// Functions/Image Filtering/F_VN_FillHoles

	{attribute 'TcIecLibraryType'}
	{attribute 'external_name' := 'F_VN_FillHoles_GUID_45C31AD9_EBC0_4725_EDA8_84DF2214AC65'}
	(* Fill holes within a gray-scale single-channel image. (equivalent to finding dark border objects) *)
	FUNCTION F_VN_FillHoles : HRESULT
	VAR_INPUT
		ipSrcImage	:	ITcVnImage;	(* Source image (USINT, UINT, INT, REAL, or LREAL, 1 channel) *)
		ipDestImage	:	REFERENCE TO ITcVnImage;	(* Destination image (An appropriate destination image will be created if required.) *)
		hrPrev	:	HRESULT;	(* HRESULT indicating the result of previous operations (If SUCCEEDED(hrPrev) equals false, no operation is executed.) *)
	END_VAR

END_FUNCTION

// Functions/Image Filtering/F_VN_GaussianFilter

	{attribute 'TcIecLibraryType'}
	{attribute 'external_name' := 'F_VN_GaussianFilter_GUID_95A7A389_C35E_4A28_C080_30D43CAAA1FC'}
	(* Apply a Gaussian filter to smooth the image. *)
	FUNCTION F_VN_GaussianFilter : HRESULT
	VAR_INPUT
		ipSrcImage	:	ITcVnImage;	(* Source image *)
		ipDestImage	:	REFERENCE TO ITcVnImage;	(* Destination image (An appropriate destination image will be created if required.) *)
		nFilterWidth	:	UDINT;	(* Filter width in pixels (1, 3, 5, 7, ...) *)
		nFilterHeight	:	UDINT;	(* Filter height in pixels (1, 3, 5, 7, ...) *)
		hrPrev	:	HRESULT;	(* HRESULT indicating the result of previous operations (If SUCCEEDED(hrPrev) equals false, no operation is executed.) *)
	END_VAR

END_FUNCTION

// Functions/Image Filtering/F_VN_GaussianFilterExp

	{attribute 'TcIecLibraryType'}
	{attribute 'external_name' := 'F_VN_GaussianFilterExp_GUID_44AEB57C_BFD9_4E61_C3CD_471B6E3D0B02'}
	(* Apply a Gaussian filter to smooth the image. (expert function) *)
	FUNCTION F_VN_GaussianFilterExp : HRESULT
	VAR_INPUT
		ipSrcImage	:	ITcVnImage;	(* Source image *)
		ipDestImage	:	REFERENCE TO ITcVnImage;	(* Destination image (An appropriate destination image will be created if required.) *)
		nFilterWidth	:	UDINT;	(* Filter width in pixels (1, 3, 5, 7, ...) *)
		nFilterHeight	:	UDINT;	(* Filter height in pixels (1, 3, 5, 7, ...) *)
		fSigmaX	:	LREAL;	(* Gaussian kernel standard deviation in X direction (>= 0, automatically chosen if 0) *)
		fSigmaY	:	LREAL;	(* Gaussian kernel standard deviation in Y direction (>= 0, automatically chosen if 0) *)
		eBorderType	:	ETcVnBorderInterpolationMethod;	(* Image border handling *)
		hrPrev	:	HRESULT;	(* HRESULT indicating the result of previous operations (If SUCCEEDED(hrPrev) equals false, no operation is executed.) *)
	END_VAR

END_FUNCTION

// Functions/Image Filtering/F_VN_LaplacianFilter

	{attribute 'TcIecLibraryType'}
	{attribute 'external_name' := 'F_VN_LaplacianFilter_GUID_22F6738F_8883_4E9E_FB58_F8CB0A9D323F'}
	(* Apply a Laplacian filter to an image. *)
	FUNCTION F_VN_LaplacianFilter : HRESULT
	VAR_INPUT
		ipSrcImage	:	ITcVnImage;	(* Source image *)
		ipDestImage	:	REFERENCE TO ITcVnImage;	(* Destination image (An appropriate destination image will be created if required.) *)
		eDestDepth	:	ETcVnElementType;	(* Destination image depth *)
		hrPrev	:	HRESULT;	(* HRESULT indicating the result of previous operations (If SUCCEEDED(hrPrev) equals false, no operation is executed.) *)
	END_VAR

END_FUNCTION

// Functions/Image Filtering/F_VN_LaplacianFilterExp

	{attribute 'TcIecLibraryType'}
	{attribute 'external_name' := 'F_VN_LaplacianFilterExp_GUID_80C0BC32_CA68_4BC2_FC4E_748676C48192'}
	(* Apply a Laplacian filter to an image. (expert function) *)
	FUNCTION F_VN_LaplacianFilterExp : HRESULT
	VAR_INPUT
		ipSrcImage	:	ITcVnImage;	(* Source image *)
		ipDestImage	:	REFERENCE TO ITcVnImage;	(* Destination image (An appropriate destination image will be created if required.) *)
		eDestDepth	:	ETcVnElementType;	(* Destination image depth *)
		nKernelSize	:	UDINT;	(* Aperture size used to compute the second-derivative filters (1, 3, 5, ..., 31) *)
		fScale	:	LREAL;	(* Scale factor for the computed derivative values *)
		fDelta	:	LREAL;	(* Delta value that is added to the results before storing them *)
		eBorderType	:	ETcVnBorderInterpolationMethod;	(* Image border handling *)
		hrPrev	:	HRESULT;	(* HRESULT indicating the result of previous operations (If SUCCEEDED(hrPrev) equals false, no operation is executed.) *)
	END_VAR

END_FUNCTION

// Functions/Image Filtering/F_VN_LocalMaxima

	{attribute 'TcIecLibraryType'}
	{attribute 'external_name' := 'F_VN_LocalMaxima_GUID_037C572B_82DC_43A0_C6A2_016E37C2D982'}
	(* Find local maxima in a gray-scale single-channel image. The found maxima are marked by a value of 1 in the destination image. *)
	FUNCTION F_VN_LocalMaxima : HRESULT
	VAR_INPUT
		ipSrcImage	:	ITcVnImage;	(* Source image (USINT or UINT, 1 channel) *)
		ipDestImage	:	REFERENCE TO ITcVnImage;	(* Destination image (Must be different from ipSrcImage! An appropriate destination image will be created if required.) *)
		hrPrev	:	HRESULT;	(* HRESULT indicating the result of previous operations (If SUCCEEDED(hrPrev) equals false, no operation is executed.) *)
	END_VAR

END_FUNCTION

// Functions/Image Filtering/F_VN_LocalMinima

	{attribute 'TcIecLibraryType'}
	{attribute 'external_name' := 'F_VN_LocalMinima_GUID_332C39B6_195E_4830_D66F_8C7BE687196D'}
	(* Find local minima in a gray-scale single-channel image. The found minima are marked by a value of 1 in the destination image. *)
	FUNCTION F_VN_LocalMinima : HRESULT
	VAR_INPUT
		ipSrcImage	:	ITcVnImage;	(* Source image (USINT or UINT, 1 channel) *)
		ipDestImage	:	REFERENCE TO ITcVnImage;	(* Destination image (Must be different from ipSrcImage! An appropriate destination image will be created if required.) *)
		hrPrev	:	HRESULT;	(* HRESULT indicating the result of previous operations (If SUCCEEDED(hrPrev) equals false, no operation is executed.) *)
	END_VAR

END_FUNCTION

// Functions/Image Filtering/F_VN_MedianFilter

	{attribute 'TcIecLibraryType'}
	{attribute 'external_name' := 'F_VN_MedianFilter_GUID_183F28CD_813D_43D0_CDC8_13AA290F7025'}
	(* Apply a Median filter to an image. *)
	FUNCTION F_VN_MedianFilter : HRESULT
	VAR_INPUT
		ipSrcImage	:	ITcVnImage;	(* Source image (for nFilterSize 3 or 5: USINT, UINT, REAL. For bigger filters, only USINT is supported. *)
		ipDestImage	:	REFERENCE TO ITcVnImage;	(* Destination image (An appropriate destination image will be created if required.) *)
		nFilterSize	:	UDINT;	(* Size (width and height) of the filter (3, 5, 7, ...) *)
		hrPrev	:	HRESULT;	(* HRESULT indicating the result of previous operations (If SUCCEEDED(hrPrev) equals false, no operation is executed.) *)
	END_VAR

END_FUNCTION

// Functions/Image Filtering/F_VN_MorphologicalOperator

	{attribute 'TcIecLibraryType'}
	{attribute 'external_name' := 'F_VN_MorphologicalOperator_GUID_B23434BD_E36C_4E02_E145_B2ED6C6CC2A2'}
	(* Apply a morphological operator. *)
	FUNCTION F_VN_MorphologicalOperator : HRESULT
	VAR_INPUT
		ipSrcImage	:	ITcVnImage;	(* Source image (only 1 channel supported for reconstruction operators) *)
		ipDestImage	:	REFERENCE TO ITcVnImage;	(* Destination image (An appropriate destination image will be created if required.) *)
		eOperator	:	ETcVnMorphologicalOperator;	(* Operator type *)
		ipStructuringElement	:	ITcVnImage;	(* Structuring element to be applied (Typically created via F_VN_CreateStructuringElement.) *)
		hrPrev	:	HRESULT;	(* HRESULT indicating the result of previous operations (If SUCCEEDED(hrPrev) equals false, no operation is executed.) *)
	END_VAR

END_FUNCTION

// Functions/Image Filtering/F_VN_RemoveLocalMaxima

	{attribute 'TcIecLibraryType'}
	{attribute 'external_name' := 'F_VN_RemoveLocalMaxima_GUID_63A5ADDB_B6C9_4B05_E1FA_40A640049502'}
	(* Remove local maxima up to a given height from a gray-scale single-channel image. *)
	FUNCTION F_VN_RemoveLocalMaxima : HRESULT
	VAR_INPUT
		ipSrcImage	:	ITcVnImage;	(* Source image (USINT, UINT, INT, REAL, or LREAL, 1 channel) *)
		ipDestImage	:	REFERENCE TO ITcVnImage;	(* Destination image (An appropriate destination image will be created if required.) *)
		fHeight	:	LREAL;	(* Maximum height of the maxima to be removed (must be greater than 0) *)
		hrPrev	:	HRESULT;	(* HRESULT indicating the result of previous operations (If SUCCEEDED(hrPrev) equals false, no operation is executed.) *)
	END_VAR

END_FUNCTION

// Functions/Image Filtering/F_VN_RemoveLocalMinima

	{attribute 'TcIecLibraryType'}
	{attribute 'external_name' := 'F_VN_RemoveLocalMinima_GUID_D50AAA78_D3B9_408D_D404_A332605EC262'}
	(* Remove local minima up to a given height from a gray-scale single-channel image. *)
	FUNCTION F_VN_RemoveLocalMinima : HRESULT
	VAR_INPUT
		ipSrcImage	:	ITcVnImage;	(* Source image (USINT, UINT, INT, REAL, or LREAL, 1 channel) *)
		ipDestImage	:	REFERENCE TO ITcVnImage;	(* Destination image (An appropriate destination image will be created if required.) *)
		fHeight	:	LREAL;	(* Maximum height of the minima to be removed (must be greater than 0) *)
		hrPrev	:	HRESULT;	(* HRESULT indicating the result of previous operations (If SUCCEEDED(hrPrev) equals false, no operation is executed.) *)
	END_VAR

END_FUNCTION

// Functions/Image Filtering/F_VN_ScharrFilter

	{attribute 'TcIecLibraryType'}
	{attribute 'external_name' := 'F_VN_ScharrFilter_GUID_4C4A4FDA_AE3C_464A_CF07_94424B3EAEFE'}
	(* Calculates the first order derivative in x or y direction using a Scharr filter. *)
	FUNCTION F_VN_ScharrFilter : HRESULT
	VAR_INPUT
		ipSrcImage	:	ITcVnImage;	(* Source image *)
		ipDestImage	:	REFERENCE TO ITcVnImage;	(* Destination image (An appropriate destination image will be created if required.) *)
		eDestDepth	:	ETcVnElementType;	(* Destination image depth *)
		eFilterDirection	:	ETcVnFilterDirection;	(* Filter direction *)
		hrPrev	:	HRESULT;	(* HRESULT indicating the result of previous operations (If SUCCEEDED(hrPrev) equals false, no operation is executed.) *)
	END_VAR

END_FUNCTION

// Functions/Image Filtering/F_VN_ScharrFilterExp

	{attribute 'TcIecLibraryType'}
	{attribute 'external_name' := 'F_VN_ScharrFilterExp_GUID_6408ADDC_C84A_4DA3_CB0C_8C03DB762CD6'}
	(* Calculates the first order derivative in x or y direction using a Scharr filter. (expert function) *)
	FUNCTION F_VN_ScharrFilterExp : HRESULT
	VAR_INPUT
		ipSrcImage	:	ITcVnImage;	(* Source image *)
		ipDestImage	:	REFERENCE TO ITcVnImage;	(* Destination image (An appropriate destination image will be created if required.) *)
		eDestDepth	:	ETcVnElementType;	(* Destination image depth *)
		eFilterDirection	:	ETcVnFilterDirection;	(* Filter direction *)
		fScale	:	LREAL;	(* Scale factor for the computed derivative values *)
		fDelta	:	LREAL;	(* Delta value that is added to the results prior to storing them in dest *)
		eBorderType	:	ETcVnBorderInterpolationMethod;	(* Image border handling *)
		hrPrev	:	HRESULT;	(* HRESULT indicating the result of previous operations (If SUCCEEDED(hrPrev) equals false, no operation is executed.) *)
	END_VAR

END_FUNCTION

// Functions/Image Filtering/F_VN_SeparableCustomFilter

	{attribute 'TcIecLibraryType'}
	{attribute 'external_name' := 'F_VN_SeparableCustomFilter_GUID_1310DFB7_D59D_44ED_EDCE_83E1B6FDCC84'}
	(* Apply a separable custom filter to the image. *)
	FUNCTION F_VN_SeparableCustomFilter : HRESULT
	VAR_INPUT
		ipSrcImage	:	ITcVnImage;	(* Source image *)
		ipDestImage	:	REFERENCE TO ITcVnImage;	(* Destination image (An appropriate destination image will be created if required.) *)
		eDestDepth	:	ETcVnElementType;	(* Destination image depth *)
	END_VAR
	VAR_IN_OUT
		stKernelX	:	TcVnMatrix;	(* 1D custom row-filter kernel with values of type REAL or LREAL *)
		stKernelY	:	TcVnMatrix;	(* 1D custom column-filter kernel with values of type REAL or LREAL *)
	END_VAR
	VAR_INPUT
		hrPrev	:	HRESULT;	(* HRESULT indicating the result of previous operations (If SUCCEEDED(hrPrev) equals false, no operation is executed.) *)
	END_VAR

END_FUNCTION

// Functions/Image Filtering/F_VN_SeparableCustomFilterExp

	{attribute 'TcIecLibraryType'}
	{attribute 'external_name' := 'F_VN_SeparableCustomFilterExp_GUID_BCC4F12D_D44C_4679_C6D6_F7CE17C8407A'}
	(* Apply a separable custom filter to the image. (expert function) *)
	FUNCTION F_VN_SeparableCustomFilterExp : HRESULT
	VAR_INPUT
		ipSrcImage	:	ITcVnImage;	(* Source image *)
		ipDestImage	:	REFERENCE TO ITcVnImage;	(* Destination image (An appropriate destination image will be created if required.) *)
		eDestDepth	:	ETcVnElementType;	(* Destination image depth *)
	END_VAR
	VAR_IN_OUT
		stKernelX	:	TcVnMatrix;	(* 1D custom row-filter kernel with values of type REAL or LREAL *)
		stKernelY	:	TcVnMatrix;	(* 1D custom column-filter kernel with values of type REAL or LREAL *)
		aAnchor	:	TcVnPoint;	(* Anchor point of the kernel *)
	END_VAR
	VAR_INPUT
		fDelta	:	LREAL;	(* Value added to each pixel after filtering *)
		eBorderType	:	ETcVnBorderInterpolationMethod;	(* Image border handling *)
		hrPrev	:	HRESULT;	(* HRESULT indicating the result of previous operations (If SUCCEEDED(hrPrev) equals false, no operation is executed.) *)
	END_VAR

END_FUNCTION

// Functions/Image Filtering/F_VN_SobelFilter

	{attribute 'TcIecLibraryType'}
	{attribute 'external_name' := 'F_VN_SobelFilter_GUID_082961EA_2A54_4C56_CFFB_604B528A29B1'}
	(* Calculates the first, second, or mixed image derivatives using an extended Sobel filter. *)
	FUNCTION F_VN_SobelFilter : HRESULT
	VAR_INPUT
		ipSrcImage	:	ITcVnImage;	(* Source image *)
		ipDestImage	:	REFERENCE TO ITcVnImage;	(* Destination image (An appropriate destination image will be created if required.) *)
		eDestDepth	:	ETcVnElementType;	(* Destination image depth *)
		nXOrder	:	UDINT;	(* Order of the x-derivative (0, 1, 2) *)
		nYOrder	:	UDINT;	(* Order of the y-derivative (0, 1, 2) *)
		hrPrev	:	HRESULT;	(* HRESULT indicating the result of previous operations (If SUCCEEDED(hrPrev) equals false, no operation is executed.) *)
	END_VAR

END_FUNCTION

// Functions/Image Filtering/F_VN_SobelFilterExp

	{attribute 'TcIecLibraryType'}
	{attribute 'external_name' := 'F_VN_SobelFilterExp_GUID_8B414AB6_412D_41C9_E4E5_57ECB320A706'}
	(* Calculates the first, second, third, or mixed image derivatives using an extended Sobel filter. (expert function) *)
	FUNCTION F_VN_SobelFilterExp : HRESULT
	VAR_INPUT
		ipSrcImage	:	ITcVnImage;	(* Source image *)
		ipDestImage	:	REFERENCE TO ITcVnImage;	(* Destination image (An appropriate destination image will be created if required.) *)
		eDestDepth	:	ETcVnElementType;	(* Destination image depth *)
		nXOrder	:	UDINT;	(* Order of the x-derivative (must be < nKernelSize) *)
		nYOrder	:	UDINT;	(* Order of the y-derivative (must be < nKernelSize) *)
		nKernelSize	:	UDINT;	(* Size of the extended Sobel kernel (3, 5, 7, ..., 31) *)
		fScale	:	LREAL;	(* Scale factor for the computed derivative values *)
		fDelta	:	LREAL;	(* Delta value that is added to the results prior to storing them in dest *)
		eBorderType	:	ETcVnBorderInterpolationMethod;	(* Image border handling *)
		hrPrev	:	HRESULT;	(* HRESULT indicating the result of previous operations (If SUCCEEDED(hrPrev) equals false, no operation is executed.) *)
	END_VAR

END_FUNCTION

// Functions/Image Filtering/F_VN_VarianceFilter

	{attribute 'TcIecLibraryType'}
	{attribute 'external_name' := 'F_VN_VarianceFilter_GUID_02C328AD_BE75_4B70_DC76_31CB3237B1CA'}
	(* Calculates the local variance of an image. *)
	FUNCTION F_VN_VarianceFilter : HRESULT
	VAR_INPUT
		ipSrcImage	:	ITcVnImage;	(* Source image. Only TCVN_ET_USINT Type is supported.  *)
		ipDestImage	:	REFERENCE TO ITcVnImage;	(* Destination image of type TCVN_ET_UINT (An appropriate destination image will be created if required.) *)
		nKernelSize	:	UDINT;	(* Size of the kernel *)
		hrPrev	:	HRESULT;	(* HRESULT indicating the result of previous operations (If SUCCEEDED(hrPrev) equals false, no operation is executed.) *)
	END_VAR

END_FUNCTION

// Functions/Image Filtering/F_VN_VarianceFilterExp

	{attribute 'TcIecLibraryType'}
	{attribute 'external_name' := 'F_VN_VarianceFilterExp_GUID_48CB282B_6C36_4355_F8DD_C52CAA374075'}
	(* Calculates the local variance of an image. (expert function) *)
	FUNCTION F_VN_VarianceFilterExp : HRESULT
	VAR_INPUT
		ipSrcImage	:	ITcVnImage;	(* Source image. Only TCVN_ET_USINT Type is supported. *)
		ipDestImage	:	REFERENCE TO ITcVnImage;	(* Destination image of type TCVN_ET_UINT (An appropriate destination image will be created if required.) *)
		nKernelSize	:	UDINT;	(* Size of the kernel *)
		fScale	:	LREAL;	(* Scale factor for the computed variance values *)
		eBorderType	:	ETcVnBorderInterpolationMethod;	(* Image border handling *)
		hrPrev	:	HRESULT;	(* HRESULT indicating the result of previous operations (If SUCCEEDED(hrPrev) equals false, no operation is executed.) *)
	END_VAR

END_FUNCTION

// Functions/Miscellaneous/F_VN_CheckFunctionInitialization

	{attribute 'TcIecLibraryType'}
	{attribute 'external_name' := 'F_VN_CheckFunctionInitialization_GUID_2C8223A2_77FF_41C2_DA7B_831BEC82D7D0'}
	(* Check if a function is initialized with the specified options. *)
	FUNCTION F_VN_CheckFunctionInitialization : HRESULT
	VAR_INPUT
		eFunction	:	ETcVnInitializableFunction;	(* Initializable function *)
		nOptions	:	ULINT;	(* Initialization options for the function *)
		hrPrev	:	HRESULT;	(* HRESULT indicating the result of previous operations (If SUCCEEDED(hrPrev) equals false, no operation is executed.) *)
	END_VAR

END_FUNCTION

// Functions/Miscellaneous/F_VN_ClipLineToBoundary

	{attribute 'TcIecLibraryType'}
	{attribute 'external_name' := 'F_VN_ClipLineToBoundary_GUID_B482B9AE_8531_4446_C981_B7F9A09BE1A0'}
	(* Clips a line to a rectangular boundary. *)
	FUNCTION F_VN_ClipLineToBoundary : HRESULT
	VAR_IN_OUT
		aLine	:	TcVnVector4_LREAL;	(* The first and second element describe the x and y component of the direction vector. The third and fourth element describe the x and y component of the position vector. *)
	END_VAR
	VAR_INPUT
		nX1	:	DINT;	(* x of top left rectangle point *)
		nY1	:	DINT;	(* y of top left rectangle point *)
		nX2	:	DINT;	(* x of bottom right rectangle point *)
		nY2	:	DINT;	(* Y of bottom right rectangle point *)
	END_VAR
	VAR_IN_OUT
		aStartPoint	:	TcVnPoint2_REAL;	(* Returns the clipped starting point of the line. *)
		aEndPoint	:	TcVnPoint2_REAL;	(* Returns the clipped end point of the line. *)
	END_VAR
	VAR_INPUT
		hrPrev	:	HRESULT;	(* HRESULT indicating the result of previous operations (If SUCCEEDED(hrPrev) equals false, no operation is executed.) *)
	END_VAR

END_FUNCTION

// Functions/Miscellaneous/F_VN_ClipLineToBoundary_ITcVnImage

	{attribute 'TcIecLibraryType'}
	{attribute 'external_name' := 'F_VN_ClipLineToBoundary_ITcVnImage_GUID_0FCA2B5E_8797_43C5_D314_057DDEA9B856'}
	(* Clips a line to the boundary of an image. *)
	FUNCTION F_VN_ClipLineToBoundary_ITcVnImage : HRESULT
	VAR_IN_OUT
		aLine	:	TcVnVector4_LREAL;	(* The first and second element describe the x and y component of the direction vector. The third and fourth element describe the x and y component of the position vector. *)
	END_VAR
	VAR_INPUT
		ipImage	:	ITcVnImage;	(* Image, from which to derive the boundary *)
	END_VAR
	VAR_IN_OUT
		aStartPoint	:	TcVnPoint2_REAL;	(* Returns the clipped starting point of the line. *)
		aEndPoint	:	TcVnPoint2_REAL;	(* Returns the clipped end point of the line. *)
	END_VAR
	VAR_INPUT
		hrPrev	:	HRESULT;	(* HRESULT indicating the result of previous operations (If SUCCEEDED(hrPrev) equals false, no operation is executed.) *)
	END_VAR

END_FUNCTION

// Functions/Miscellaneous/F_VN_ClipLineToBoundary_TcVnRectangle_DINT

	{attribute 'TcIecLibraryType'}
	{attribute 'external_name' := 'F_VN_ClipLineToBoundary_TcVnRectangle_DINT_GUID_6C0A9627_1BE4_42B6_C7E1_34156AEEC835'}
	(* Clips a line to a rectangular boundary. *)
	FUNCTION F_VN_ClipLineToBoundary_TcVnRectangle_DINT : HRESULT
	VAR_IN_OUT
		aLine	:	TcVnVector4_LREAL;	(* The first and second element describe the x and y component of the direction vector. The third and fourth element describe the x and y component of the position vector. *)
		stRectangle	:	TcVnRectangle_DINT;	(* Rectangular boundary *)
		aStartPoint	:	TcVnPoint2_REAL;	(* Returns the clipped starting point of the line. *)
		aEndPoint	:	TcVnPoint2_REAL;	(* Returns the clipped end point of the line. *)
	END_VAR
	VAR_INPUT
		hrPrev	:	HRESULT;	(* HRESULT indicating the result of previous operations (If SUCCEEDED(hrPrev) equals false, no operation is executed.) *)
	END_VAR

END_FUNCTION

// Functions/Miscellaneous/F_VN_ConvertITcUnknownToITcVnBitmapExport

	{attribute 'TcIecLibraryType'}
	{attribute 'external_name' := 'F_VN_ConvertITcUnknownToITcVnBitmapExport_GUID_C5AC5150_1991_4233_D664_F885FA18923A'}
	(* Convert an ITcUnknown interface pointer to an ITcVnBitmapExport interface pointer. The destination pointer will be released (if existing) and set to the source pointer. The source pointer will be set to 0. *)
	FUNCTION F_VN_ConvertITcUnknownToITcVnBitmapExport : HRESULT
	VAR_INPUT
		ipSrc	:	REFERENCE TO ITcUnknown;	(* Source pointer *)
		ipDest	:	REFERENCE TO ITcVnBitmapExport;	(* Destination pointer *)
		hrPrev	:	HRESULT;	(* HRESULT indicating the result of previous operations (If SUCCEEDED(hrPrev) equals false, no operation is executed.) *)
	END_VAR

END_FUNCTION

// Functions/Miscellaneous/F_VN_ConvertITcUnknownToITcVnContainer

	{attribute 'TcIecLibraryType'}
	{attribute 'external_name' := 'F_VN_ConvertITcUnknownToITcVnContainer_GUID_F89008A1_7EE5_44B8_ED7B_BAB16CAC9C5B'}
	(* Convert an ITcUnknown interface pointer to an ITcVnContainer interface pointer. The destination pointer will be released (if existing) and set to the source pointer. The source pointer will be set to 0. *)
	FUNCTION F_VN_ConvertITcUnknownToITcVnContainer : HRESULT
	VAR_INPUT
		ipSrc	:	REFERENCE TO ITcUnknown;	(* Source pointer *)
		ipDest	:	REFERENCE TO ITcVnContainer;	(* Destination pointer *)
		hrPrev	:	HRESULT;	(* HRESULT indicating the result of previous operations (If SUCCEEDED(hrPrev) equals false, no operation is executed.) *)
	END_VAR

END_FUNCTION

// Functions/Miscellaneous/F_VN_ConvertITcUnknownToITcVnImage

	{attribute 'TcIecLibraryType'}
	{attribute 'external_name' := 'F_VN_ConvertITcUnknownToITcVnImage_GUID_F768478E_506F_4CE2_C2D1_8F48D5018F3E'}
	(* Convert an ITcUnknown interface pointer to an ITcVnImage interface pointer. The destination pointer will be released (if existing) and set to the source pointer. The source pointer will be set to 0. *)
	FUNCTION F_VN_ConvertITcUnknownToITcVnImage : HRESULT
	VAR_INPUT
		ipSrc	:	REFERENCE TO ITcUnknown;	(* Source pointer *)
		ipDest	:	REFERENCE TO ITcVnImage;	(* Destination pointer *)
		hrPrev	:	HRESULT;	(* HRESULT indicating the result of previous operations (If SUCCEEDED(hrPrev) equals false, no operation is executed.) *)
	END_VAR

END_FUNCTION

// Functions/Miscellaneous/F_VN_ConvertITcUnknownToITcVnMlModel

	{attribute 'TcIecLibraryType'}
	{attribute 'external_name' := 'F_VN_ConvertITcUnknownToITcVnMlModel_GUID_EBE69EF4_1DE6_4A53_D37C_0D2CB88EB72B'}
	(* Convert an ITcUnknown interface pointer to an ITcVnMlModel interface pointer. The destination pointer will be released (if existing) and set to the source pointer. The source pointer will be set to 0. *)
	FUNCTION F_VN_ConvertITcUnknownToITcVnMlModel : HRESULT
	VAR_INPUT
		ipSrc	:	REFERENCE TO ITcUnknown;	(* Source pointer *)
		ipDest	:	REFERENCE TO ITcVnMlModel;	(* Destination pointer *)
		hrPrev	:	HRESULT;	(* HRESULT indicating the result of previous operations (If SUCCEEDED(hrPrev) equals false, no operation is executed.) *)
	END_VAR

END_FUNCTION

// Functions/Miscellaneous/F_VN_DeinitializeFunction

	{attribute 'TcIecLibraryType'}
	{attribute 'external_name' := 'F_VN_DeinitializeFunction_GUID_D1F3361E_3ED0_4425_EAC1_FD419D650FCA'}
	(* Deinitialize the specified options for the function. *)
	FUNCTION F_VN_DeinitializeFunction : HRESULT
	VAR_INPUT
		eFunction	:	ETcVnInitializableFunction;	(* Initializable function *)
		nOptions	:	ULINT;	(* Initialization options for the function *)
		hrPrev	:	HRESULT;	(* HRESULT indicating the result of previous operations (If SUCCEEDED(hrPrev) equals false, no operation is executed.) *)
	END_VAR

END_FUNCTION

// Functions/Miscellaneous/F_VN_GetTimestamp

	{attribute 'TcIecLibraryType'}
	{attribute 'external_name' := 'F_VN_GetTimestamp_GUID_2D68E61A_B781_405D_F127_30855B02D50E'}
	(* Get the timestamp (actual DC time) from the last change of an object (e.g. ITcVnImage or ITcVnContainer) *)
	FUNCTION F_VN_GetTimestamp : HRESULT
	VAR_INPUT
		ipUnknown	:	ITcUnknown;	(* An object implementing ITcUnknown and ITcVnTimestamp (e.g. ITcVnImage or ITcVnContainer) *)
	END_VAR
	VAR_IN_OUT
		nTimestamp	:	LINT;	(* Returns the timestamp *)
	END_VAR
	VAR_INPUT
		hrPrev	:	HRESULT;	(* HRESULT indicating the result of previous operations (If SUCCEEDED(hrPrev) equals false, no operation is executed.) *)
	END_VAR

END_FUNCTION

// Functions/Miscellaneous/F_VN_HuMomentInvariants

	{attribute 'TcIecLibraryType'}
	{attribute 'external_name' := 'F_VN_HuMomentInvariants_GUID_578FD112_2DC5_4CAD_F1B3_F670083C2AF6'}
	(* Computes the Hu moment invariants. *)
	FUNCTION F_VN_HuMomentInvariants : HRESULT
	VAR_IN_OUT
		stMoments	:	TcVnMoments;	(* Moments from which to compute the Hu invariants *)
		aHuInvariants	:	TcVnArray7_LREAL;	(* Returns the Hu moment invariants *)
	END_VAR
	VAR_INPUT
		hrPrev	:	HRESULT;	(* HRESULT indicating the result of previous operations (If SUCCEEDED(hrPrev) equals false, no operation is executed.) *)
	END_VAR

END_FUNCTION

// Functions/Miscellaneous/F_VN_InitMatrixStruct

	{attribute 'TcIecLibraryType'}
	{attribute 'external_name' := 'F_VN_InitMatrixStruct_GUID_6C97114E_1940_4DE0_F672_C2C518D51A5C'}
	(* Initialize a struct of the type TcVnMatrix extending a buffer with metainformation so that it can be used as a matrix. *)
	FUNCTION F_VN_InitMatrixStruct : HRESULT
	VAR_INPUT
		pSrcBuffer	:	PVOID;	(* Source buffer *)
	END_VAR
	VAR_IN_OUT
		stDestMatrix	:	TcVnMatrix;	(* Returns completed matrix struct *)
	END_VAR
	VAR_INPUT
		nRows	:	UDINT;	(* Matrix rows *)
		nCols	:	UDINT;	(* Matrix columns *)
		eElementType	:	ETcVnElementType;	(* Type of the matrix elements *)
		hrPrev	:	HRESULT;	(* HRESULT indicating the result of previous operations (If SUCCEEDED(hrPrev) equals false, no operation is executed.) *)
	END_VAR

END_FUNCTION

// Functions/Miscellaneous/F_VN_InvertMatrix3x3

	{attribute 'TcIecLibraryType'}
	{attribute 'external_name' := 'F_VN_InvertMatrix3x3_GUID_03AE1FC5_20A2_4AD9_CEFD_6FDE03EABABD'}
	(* Invert a 3x3 matrix. *)
	FUNCTION F_VN_InvertMatrix3x3 : HRESULT
	VAR_IN_OUT
		aSrcMatrix	:	TcVnMatrix3x3_LREAL;	(* Source matrix *)
		aInvertedMatrix	:	TcVnMatrix3x3_LREAL;	(* Returns inverted matrix *)
	END_VAR
	VAR_INPUT
		hrPrev	:	HRESULT;	(* HRESULT indicating the result of previous operations (If SUCCEEDED(hrPrev) equals false, no operation is executed.) *)
	END_VAR

END_FUNCTION

// Functions/Miscellaneous/F_VN_LineIntersectionPoint

	{attribute 'TcIecLibraryType'}
	{attribute 'external_name' := 'F_VN_LineIntersectionPoint_GUID_E2C1B61F_0556_492A_F95A_4500588117C8'}
	(* Computes the intersection point between two lines (returns S_FALSE if the provided lines are parallel). *)
	FUNCTION F_VN_LineIntersectionPoint : HRESULT
	VAR_IN_OUT
		aLine1	:	TcVnVector4_LREAL;	(* First line. The first and second element describe the x and y component of a vector collinear to the line. The third and fourth element describe the x and y component of a point on the line. *)
		aLine2	:	TcVnVector4_LREAL;	(* Second line. The first and second element describe the x and y component of a vector collinear to the line. The third and fourth element describe the x and y component of a point on the line. *)
		aIntersecPoint	:	TcVnPoint2_REAL;	(* Returns the intersection point of aLine1 and aLine2. *)
	END_VAR
	VAR_INPUT
		hrPrev	:	HRESULT;	(* HRESULT indicating the result of previous operations (If SUCCEEDED(hrPrev) equals false, no operation is executed.) *)
	END_VAR

END_FUNCTION

// Functions/Miscellaneous/F_VN_LineIntersectionPointAndAngle

	{attribute 'TcIecLibraryType'}
	{attribute 'external_name' := 'F_VN_LineIntersectionPointAndAngle_GUID_E9B34839_7FE9_48FF_FE7B_BB862FD5C3F1'}
	(* Computes the intersection point and angle between two lines (returns S_FALSE if the provided lines are parallel). *)
	FUNCTION F_VN_LineIntersectionPointAndAngle : HRESULT
	VAR_IN_OUT
		aLine1	:	TcVnVector4_LREAL;	(* First line. The first and second element describe the x and y component of a vector collinear to the line. The third and fourth element describe the x and y component of a point on the line. *)
		aLine2	:	TcVnVector4_LREAL;	(* Second line. The first and second element describe the x and y component of a vector collinear to the line. The third and fourth element describe the x and y component of a point on the line. *)
		aIntersecPoint	:	TcVnPoint2_REAL;	(* Returns the intersection point of aLine1 and aLine2. *)
		fAngle	:	REAL;	(* Returns the intersection angle of aLine1 and aLine2. *)
	END_VAR
	VAR_INPUT
		bAngleInDegrees	:	BOOL;	(* If TRUE, fAngle is in degrees. If FALSE, fAngle is in radians. *)
		hrPrev	:	HRESULT;	(* HRESULT indicating the result of previous operations (If SUCCEEDED(hrPrev) equals false, no operation is executed.) *)
	END_VAR

END_FUNCTION

// Functions/Miscellaneous/F_VN_MultiplyMatrices

	{attribute 'TcIecLibraryType'}
	{attribute 'external_name' := 'F_VN_MultiplyMatrices_GUID_054449C6_10D9_4AE6_FA2D_654136AF7B74'}
	(* Matrix multiplication of two matrices (A * B = C). All matrices are represented by structs holding a pointer to an array of the appropriate size. *)
	FUNCTION F_VN_MultiplyMatrices : HRESULT
	VAR_IN_OUT
		stSrcMatrix1	:	TcVnMatrix;	(* First source matrix (A) *)
		stSrcMatrix2	:	TcVnMatrix;	(* Second source matrix (B) *)
		stDestMatrix	:	TcVnMatrix;	(* Destination matrix (C) (The destination matrix is filled by this function, but the required memory needs to be provided.) *)
	END_VAR
	VAR_INPUT
		hrPrev	:	HRESULT;	(* HRESULT indicating the result of previous operations (If SUCCEEDED(hrPrev) equals false, no operation is executed.) *)
	END_VAR

END_FUNCTION

// Functions/Miscellaneous/F_VN_RotatedRectangleCorners

	{attribute 'TcIecLibraryType'}
	{attribute 'external_name' := 'F_VN_RotatedRectangleCorners_GUID_D92E77CB_99B2_4A0D_E11B_9DA419F9BEA0'}
	(* Computes the 4 corner points of a rotated rectangle. *)
	FUNCTION F_VN_RotatedRectangleCorners : HRESULT
	VAR_IN_OUT
		stRect	:	TcVnRotatedRectangle;	(* Rotated rectangle *)
		aCorners	:	TcVnArray4_Point2_REAL;	(* Returns the 4 corner points *)
	END_VAR
	VAR_INPUT
		hrPrev	:	HRESULT;	(* HRESULT indicating the result of previous operations (If SUCCEEDED(hrPrev) equals false, no operation is executed.) *)
	END_VAR

END_FUNCTION

// Functions/Miscellaneous/F_VN_RotatedRectangleIntersection

	{attribute 'TcIecLibraryType'}
	{attribute 'external_name' := 'F_VN_RotatedRectangleIntersection_GUID_7460E821_B7CE_4696_E78E_CC91BD652AB6'}
	(* Finds the intersection of 2 rotated rectangles. *)
	FUNCTION F_VN_RotatedRectangleIntersection : HRESULT
	VAR_IN_OUT
		stRect1	:	TcVnRotatedRectangle;	(* Rotated rectangle 1 *)
		stRect2	:	TcVnRotatedRectangle;	(* Rotated rectangle 2 *)
	END_VAR
	VAR_INPUT
		ipIntersection	:	REFERENCE TO ITcVnContainer;	(* Returns the intersection points (ContainerType_Vector_TcVnPoint2_REAL, non-zero interface pointers are reused) *)
	END_VAR
	VAR_IN_OUT
		eIntersection	:	ETcVnRectangleIntersection;	(* Returns the intersection type *)
	END_VAR
	VAR_INPUT
		hrPrev	:	HRESULT;	(* HRESULT indicating the result of previous operations (If SUCCEEDED(hrPrev) equals false, no operation is executed.) *)
	END_VAR

END_FUNCTION

// Functions/Miscellaneous/F_VN_SetRngSeed

	{attribute 'TcIecLibraryType'}
	{attribute 'external_name' := 'F_VN_SetRngSeed_GUID_62925594_6E02_45A5_EFB3_4E4E3914E196'}
	(* Sets the internal pseudo random number generator seed (intended for testing purposes only). *)
	FUNCTION F_VN_SetRngSeed : HRESULT
	VAR_INPUT
		nSeed	:	DINT;	(* seed (0 sets the generator back to its initial state) *)
		hrPrev	:	HRESULT;	(* HRESULT indicating the result of previous operations (If SUCCEEDED(hrPrev) equals false, no operation is executed.) *)
	END_VAR

END_FUNCTION

// Functions/Miscellaneous/F_VN_UpdateTimestamp

	{attribute 'TcIecLibraryType'}
	{attribute 'external_name' := 'F_VN_UpdateTimestamp_GUID_B4BE518F_BCEC_4AF7_DE4A_0B9806D4C903'}
	(* Update the timestamp of an object to the actual DC time (e.g. ITcVnImage or ITcVnContainer) *)
	FUNCTION F_VN_UpdateTimestamp : HRESULT
	VAR_INPUT
		ipUnknown	:	ITcUnknown;	(* An object implementing ITcUnknown and ITcVnTimestamp (e.g. ITcVnImage or ITcVnContainer) *)
		hrPrev	:	HRESULT;	(* HRESULT indicating the result of previous operations (If SUCCEEDED(hrPrev) equals false, no operation is executed.) *)
	END_VAR

END_FUNCTION

// Functions/Basic Image Operations/F_VN_CombineImageChannels

	{attribute 'TcIecLibraryType'}
	{attribute 'external_name' := 'F_VN_CombineImageChannels_GUID_25DA3B00_18D0_46C8_E55B_F6FA19D3AC31'}
	(* Combines several single-channel images into one multi-channel image. *)
	FUNCTION F_VN_CombineImageChannels : HRESULT
	VAR_INPUT
		pSrcImages	:	PVOID;	(* Pointer to an array of single-channel source images *)
		ipDestImage	:	REFERENCE TO ITcVnImage;	(* Multi-channel destination image (An appropriate destination image will be created if required.) *)
		nSrcArraySize	:	UINT;	(* pSrcImages array size *)
		hrPrev	:	HRESULT;	(* HRESULT indicating the result of previous operations (If SUCCEEDED(hrPrev) equals false, no operation is executed.) *)
	END_VAR

END_FUNCTION

// Functions/Basic Image Operations/F_VN_ConvertElementType

	{attribute 'TcIecLibraryType'}
	{attribute 'external_name' := 'F_VN_ConvertElementType_GUID_8460C0E3_F799_4F78_CEE2_AC81B0221C55'}
	(* Converts an image to another element type. *)
	FUNCTION F_VN_ConvertElementType : HRESULT
	VAR_INPUT
		ipSrcImage	:	ITcVnImage;	(* Source image *)
		ipDestImage	:	REFERENCE TO ITcVnImage;	(* Destination image (An appropriate destination image will be created if required.) *)
		eElementType	:	ETcVnElementType;	(* Desired element type of the destination image *)
		hrPrev	:	HRESULT;	(* HRESULT indicating the result of previous operations (If SUCCEEDED(hrPrev) equals false, no operation is executed.) *)
	END_VAR

END_FUNCTION

// Functions/Basic Image Operations/F_VN_ConvertElementTypeExp

	{attribute 'TcIecLibraryType'}
	{attribute 'external_name' := 'F_VN_ConvertElementTypeExp_GUID_74975FC9_96F5_4385_D7FB_B683F33E000E'}
	(* Converts an image to another element type. (expert function) *)
	FUNCTION F_VN_ConvertElementTypeExp : HRESULT
	VAR_INPUT
		ipSrcImage	:	ITcVnImage;	(* Source image *)
		ipDestImage	:	REFERENCE TO ITcVnImage;	(* Destination image (An appropriate destination image will be created if required.) *)
		eElementType	:	ETcVnElementType;	(* Desired element type of the destination image *)
		fScaleFactor	:	LREAL;	(* Scale factor for the pixel values *)
		fDelta	:	LREAL;	(* Value that is added to the scaled pixel values *)
		hrPrev	:	HRESULT;	(* HRESULT indicating the result of previous operations (If SUCCEEDED(hrPrev) equals false, no operation is executed.) *)
	END_VAR

END_FUNCTION

// Functions/Basic Image Operations/F_VN_CopyImage

	{attribute 'TcIecLibraryType'}
	{attribute 'external_name' := 'F_VN_CopyImage_GUID_DACF2CB2_A020_460A_FD2A_D1364FE717CD'}
	(* Creates a deep copy of an image. *)
	FUNCTION F_VN_CopyImage : HRESULT
	VAR_INPUT
		ipSrcImage	:	ITcVnImage;	(* Source image *)
		ipDestImage	:	REFERENCE TO ITcVnImage;	(* Destination image (An appropriate destination image will be created if required.) *)
		hrPrev	:	HRESULT;	(* HRESULT indicating the result of previous operations (If SUCCEEDED(hrPrev) equals false, no operation is executed.) *)
	END_VAR

END_FUNCTION

// Functions/Basic Image Operations/F_VN_CopyImageRegion

	{attribute 'TcIecLibraryType'}
	{attribute 'external_name' := 'F_VN_CopyImageRegion_GUID_E3FF4DE9_BF35_44D6_CEE2_36B30039A262'}
	(* Deep copy the specified region of interest into a new image. *)
	FUNCTION F_VN_CopyImageRegion : HRESULT
	VAR_INPUT
		ipSrcImage	:	ITcVnImage;	(* Source image *)
		nX	:	UDINT;	(* Left boundary (inclusive 0-based index) *)
		nY	:	UDINT;	(* Upper boundary (inclusive 0-based index) *)
		nWidth	:	UDINT;	(* ROI width *)
		nHeight	:	UDINT;	(* ROI height *)
		ipDestImage	:	REFERENCE TO ITcVnImage;	(* Destination image (An appropriate destination image will be created if required.) *)
		hrPrev	:	HRESULT;	(* HRESULT indicating the result of previous operations (If SUCCEEDED(hrPrev) equals false, no operation is executed.) *)
	END_VAR

END_FUNCTION

// Functions/Basic Image Operations/F_VN_CopyImageRegionToRegion

	{attribute 'TcIecLibraryType'}
	{attribute 'external_name' := 'F_VN_CopyImageRegionToRegion_GUID_74D0406D_E39E_4667_E4C1_2505FF03C218'}
	(* Copy an image region into another image region. *)
	FUNCTION F_VN_CopyImageRegionToRegion : HRESULT
	VAR_INPUT
		ipSrcImage	:	ITcVnImage;	(* Source image *)
		nXSrc	:	UDINT;	(* Left boundary in ipSrcImage (inclusive 0-based index) *)
		nYSrc	:	UDINT;	(* Upper boundary in ipSrcImage (inclusive 0-based index) *)
		nWidth	:	UDINT;	(* ROI width *)
		nHeight	:	UDINT;	(* ROI height *)
		ipDestImage	:	ITcVnImage;	(* Destination image (same type as ipSrcImage) *)
		nXDest	:	UDINT;	(* Left boundary in ipDestImage (inclusive 0-based index) *)
		nYDest	:	UDINT;	(* Upper boundary in ipDestImage (inclusive 0-based index) *)
		hrPrev	:	HRESULT;	(* HRESULT indicating the result of previous operations (If SUCCEEDED(hrPrev) equals false, no operation is executed.) *)
	END_VAR

END_FUNCTION

// Functions/Basic Image Operations/F_VN_CopyIntoDisplayableImage

	{attribute 'TcIecLibraryType'}
	{attribute 'external_name' := 'F_VN_CopyIntoDisplayableImage_GUID_7045649E_D22D_4554_F804_9D96FD63DB74'}
	(* Copys an image into a displayable image. If you do not want to use ipSrcImage after this function call, you might want to use F_VN_TransformIntoDisplayableImage instead for better performance. *)
	FUNCTION F_VN_CopyIntoDisplayableImage : HRESULT
	VAR_INPUT
		ipSrcImage	:	ITcVnImage;	(* Source image *)
		ipDestImage	:	REFERENCE TO ITcVnDisplayableImage;	(* Returns the displayable image *)
		hrPrev	:	HRESULT;	(* HRESULT indicating the result of previous operations (If SUCCEEDED(hrPrev) equals false, no operation is executed.) *)
	END_VAR

END_FUNCTION

// Functions/Basic Image Operations/F_VN_TransformIntoDisplayableImage

	{attribute 'TcIecLibraryType'}
	{attribute 'external_name' := 'F_VN_TransformIntoDisplayableImage_GUID_81CBFC91_8807_4674_EF6A_E2E8664FDDC1'}
	(* Transform an image into a displayable image. The source image will be released and zeroed while existing destination images will be released and overwritten with the function result. The source image must not be used anywhere else and the transformation is very fast. If you want to use ipSrcImage after this function call, use F_VN_CopyIntoDisplayableImage instead. *)
	FUNCTION F_VN_TransformIntoDisplayableImage : HRESULT
	VAR_INPUT
		ipSrcImage	:	REFERENCE TO ITcVnImage;	(* Source image *)
		ipDestImage	:	REFERENCE TO ITcVnDisplayableImage;	(* Returns the displayable image *)
		hrPrev	:	HRESULT;	(* HRESULT indicating the result of previous operations (If SUCCEEDED(hrPrev) equals false, no operation is executed.) *)
	END_VAR

END_FUNCTION

// Functions/Basic Image Operations/F_VN_CreateAssociatedImage

	{attribute 'TcIecLibraryType'}
	{attribute 'external_name' := 'F_VN_CreateAssociatedImage_GUID_C3F8AE79_6867_4736_DA23_86359C7D10EA'}
	(* Creates a new image that shares its data with the source image. E.g. useful to work on different (disjoint) ROIs in parallel. *)
	FUNCTION F_VN_CreateAssociatedImage : HRESULT
	VAR_INPUT
		ipSrcImage	:	ITcVnImage;	(* Source image *)
		ipDestImage	:	REFERENCE TO ITcVnImage;	(* Returns the created image (Non-zero interface pointers are reused.) *)
		hrPrev	:	HRESULT;	(* HRESULT indicating the result of previous operations (If SUCCEEDED(hrPrev) equals false, no operation is executed.) *)
	END_VAR

END_FUNCTION

// Functions/Basic Image Operations/F_VN_CreateEmptyImage

	{attribute 'TcIecLibraryType'}
	{attribute 'external_name' := 'F_VN_CreateEmptyImage_GUID_04F53BCE_E9EE_4747_E504_6153C8397F99'}
	(* Creates an empty image without allocating any data buffer. The initial reference count is set to one if a new image interface is created and kept, otherwise. *)
	FUNCTION F_VN_CreateEmptyImage : HRESULT
	VAR_INPUT
		ipImage	:	REFERENCE TO ITcVnImage;	(* Returns the created image *)
		hrPrev	:	HRESULT;	(* HRESULT indicating the result of previous operations (If SUCCEEDED(hrPrev) equals false, no operation is executed.) *)
	END_VAR

END_FUNCTION

// Functions/Basic Image Operations/F_VN_CreateImage

	{attribute 'TcIecLibraryType'}
	{attribute 'external_name' := 'F_VN_CreateImage_GUID_0E5F3C04_2BBE_4FA7_D37B_E94F2B4177E2'}
	(* Creates an image and allocate an appropriate data buffer. The initial reference count is set to one if a new image interface is created and kept, otherwise. *)
	FUNCTION F_VN_CreateImage : HRESULT
	VAR_INPUT
		ipImage	:	REFERENCE TO ITcVnImage;	(* Returns the created image (Non-zero interface pointers are reused.) *)
		nWidth	:	UDINT;	(* Image width *)
		nHeight	:	UDINT;	(* Image height *)
		ePixelType	:	ETcVnElementType;	(* Pixel type *)
		nChannelNum	:	UDINT;	(* Number of channels (1 to 255) *)
		hrPrev	:	HRESULT;	(* HRESULT indicating the result of previous operations (If SUCCEEDED(hrPrev) equals false, no operation is executed.) *)
	END_VAR

END_FUNCTION

// Functions/Basic Image Operations/F_VN_CreateNDimensionalImage

	{attribute 'TcIecLibraryType'}
	{attribute 'external_name' := 'F_VN_CreateNDimensionalImage_GUID_06F11123_C16C_4CA8_DE99_AFE15FF88EB0'}
	(* Creates an N-dimensional image and allocates an appropriate data buffer. The initial reference count is set to one if a new image interface is created and kept, otherwise. *)
	FUNCTION F_VN_CreateNDimensionalImage : HRESULT
	VAR_INPUT
		ipImage	:	REFERENCE TO ITcVnImage;	(* Returns the created image (Non-zero interface pointers are reused.) *)
	END_VAR
	VAR_IN_OUT
		aShape	:	TcVnArray33_UDINT;	(* Specifies the shape of ipDestImage. First entry is the number of dimensions of ipImage (max. 32), followed by the sizes of each dimension. *)
	END_VAR
	VAR_INPUT
		ePixelType	:	ETcVnElementType;	(* Pixel type *)
		hrPrev	:	HRESULT;	(* HRESULT indicating the result of previous operations (If SUCCEEDED(hrPrev) equals false, no operation is executed.) *)
	END_VAR

END_FUNCTION

// Functions/Basic Image Operations/F_VN_CreateImageAndSetPixels

	{attribute 'TcIecLibraryType'}
	{attribute 'external_name' := 'F_VN_CreateImageAndSetPixels_GUID_2BB91321_CB18_46A8_D2E9_A9275FFCF22B'}
	(* Creates an image, allocates an appropriate data buffer and sets all pixels to the specified value. The initial reference count is set to one if a new image interface is created and kept, otherwise. *)
	FUNCTION F_VN_CreateImageAndSetPixels : HRESULT
	VAR_INPUT
		ipImage	:	REFERENCE TO ITcVnImage;	(* Returns the created image (Non-zero interface pointers are reused.) *)
		nWidth	:	UDINT;	(* Image width *)
		nHeight	:	UDINT;	(* Image height *)
		ePixelType	:	ETcVnElementType;	(* Pixel type *)
		nChannelNum	:	UDINT;	(* Number of channels (1 to 4) *)
	END_VAR
	VAR_IN_OUT
		aValue	:	TcVnVector4_LREAL;	(* Pixel value *)
	END_VAR
	VAR_INPUT
		hrPrev	:	HRESULT;	(* HRESULT indicating the result of previous operations (If SUCCEEDED(hrPrev) equals false, no operation is executed.) *)
	END_VAR

END_FUNCTION

// Functions/Basic Image Operations/F_VN_CreateNDimensionalImageAndSetPixels

	{attribute 'TcIecLibraryType'}
	{attribute 'external_name' := 'F_VN_CreateNDimensionalImageAndSetPixels_GUID_3CC8A38D_B2A8_4501_CB52_106CBCBF41F9'}
	(* Creates an N-dimensional image, allocates an appropriate data buffer and sets all pixels to the specified value. The initial reference count is set to one if a new image interface is created and kept, otherwise. *)
	FUNCTION F_VN_CreateNDimensionalImageAndSetPixels : HRESULT
	VAR_INPUT
		ipImage	:	REFERENCE TO ITcVnImage;	(* Returns the created image (Non-zero interface pointers are reused.) *)
	END_VAR
	VAR_IN_OUT
		aShape	:	TcVnArray33_UDINT;	(* Specifies the shape of ipDestImage. First entry is the number of dimensions of ipImage (max. 32), followed by the sizes of each dimension. *)
	END_VAR
	VAR_INPUT
		ePixelType	:	ETcVnElementType;	(* Pixel type *)
		fValue	:	LREAL;	(* Pixel value *)
		hrPrev	:	HRESULT;	(* HRESULT indicating the result of previous operations (If SUCCEEDED(hrPrev) equals false, no operation is executed.) *)
	END_VAR

END_FUNCTION

// Functions/Basic Image Operations/F_VN_CreateImageFromArray

	{attribute 'TcIecLibraryType'}
	{attribute 'external_name' := 'F_VN_CreateImageFromArray_GUID_E2E6C1E7_5588_4AC2_D34C_2535E5A65B84'}
	(* Creates an image and initialize it with the provided data. The initial reference count is set to one if a new image interface is created and kept, otherwise. *)
	FUNCTION F_VN_CreateImageFromArray : HRESULT
	VAR_INPUT
		pData	:	PVOID;	(* Pointer to the 1D data array. Make sure that the array contains at least nWidth * nHeight * nChannelNum elements and that the array element type matches ePixelType. *)
		ipImage	:	REFERENCE TO ITcVnImage;	(* Returns the created image (Non-zero interface pointers are reused.) *)
		nWidth	:	UDINT;	(* Image width *)
		nHeight	:	UDINT;	(* Image height *)
		ePixelType	:	ETcVnElementType;	(* Pixel type *)
		nChannelNum	:	UDINT;	(* Number of channels (1 to 255) *)
		hrPrev	:	HRESULT;	(* HRESULT indicating the result of previous operations (If SUCCEEDED(hrPrev) equals false, no operation is executed.) *)
	END_VAR

END_FUNCTION

// Functions/Basic Image Operations/F_VN_CreateNDimensionalImageFromArray

	{attribute 'TcIecLibraryType'}
	{attribute 'external_name' := 'F_VN_CreateNDimensionalImageFromArray_GUID_1CE6B49E_3821_411A_DFC2_F5460D6E1CBA'}
	(* Creates an N-dimensional image and initialize it with the provided data. The initial reference count is set to one if a new image interface is created and kept, otherwise. *)
	FUNCTION F_VN_CreateNDimensionalImageFromArray : HRESULT
	VAR_INPUT
		pData	:	PVOID;	(* Pointer to the 1D data array. Ensure that the array contains at least the number of elements equal to the product of all dimensions in aShape and that the array element type matches ePixelType. *)
		ipImage	:	REFERENCE TO ITcVnImage;	(* Returns the created image (Non-zero interface pointers are reused.) *)
	END_VAR
	VAR_IN_OUT
		aShape	:	TcVnArray33_UDINT;	(* Specifies the shape of ipDestImage. First entry is the number of dimensions of ipImage (max. 32), followed by the sizes of each dimension. *)
	END_VAR
	VAR_INPUT
		ePixelType	:	ETcVnElementType;	(* Pixel type *)
		hrPrev	:	HRESULT;	(* HRESULT indicating the result of previous operations (If SUCCEEDED(hrPrev) equals false, no operation is executed.) *)
	END_VAR

END_FUNCTION

// Functions/Basic Image Operations/F_VN_ExportImage

	{attribute 'TcIecLibraryType'}
	{attribute 'external_name' := 'F_VN_ExportImage_GUID_91B86272_4062_43A0_D8C3_6EF55FBDC4D7'}
	(* Exports the image data into a given buffer (e.g. an array). F_VN_ExportImageSize should be called before to get the required buffer size. *)
	FUNCTION F_VN_ExportImage : HRESULT
	VAR_INPUT
		ipImage	:	ITcVnImage;	(* Image *)
		pBuffer	:	PVOID;	(* Pointer to a buffer to store the image data (Make sure to allocate enough memory! The required size in bytes can be determined using the function F_VN_ExportImageSize) *)
		nBufferSize	:	ULINT;	(* Size of the buffer memory in bytes *)
		hrPrev	:	HRESULT;	(* HRESULT indicating the result of previous operations (If SUCCEEDED(hrPrev) equals false, no operation is executed.) *)
	END_VAR

END_FUNCTION

// Functions/Basic Image Operations/F_VN_ExportImageSize

	{attribute 'TcIecLibraryType'}
	{attribute 'external_name' := 'F_VN_ExportImageSize_GUID_1A071C84_B2B5_4CE3_FFA1_A89B34819B94'}
	(* Get the required buffer size (in bytes) to store the image data. *)
	FUNCTION F_VN_ExportImageSize : HRESULT
	VAR_INPUT
		ipImage	:	ITcVnImage;	(* Image *)
	END_VAR
	VAR_IN_OUT
		nBufferSize	:	ULINT;	(* Returns the required buffer size in bytes *)
	END_VAR
	VAR_INPUT
		hrPrev	:	HRESULT;	(* HRESULT indicating the result of previous operations (If SUCCEEDED(hrPrev) equals false, no operation is executed.) *)
	END_VAR

END_FUNCTION

// Functions/Basic Image Operations/F_VN_ExportImageAsBmp

	{attribute 'TcIecLibraryType'}
	{attribute 'external_name' := 'F_VN_ExportImageAsBmp_GUID_C8E1955D_94F6_4D1A_F604_D0184B1257AF'}
	(* Exports the image as bitmap into a given buffer (e.g. an array). F_VN_ExportImageAsBmpSize should be called before to get the required buffer size. *)
	FUNCTION F_VN_ExportImageAsBmp : HRESULT
	VAR_INPUT
		ipImage	:	ITcVnImage;	(* Image *)
		pBuffer	:	PVOID;	(* Pointer to a buffer to store the bitmap image (Make sure to allocate enough memory! The required size in bytes can be determined using the function F_VN_ExportImageAsBmpSize) *)
		nBufferSize	:	ULINT;	(* Size of the buffer memory in bytes *)
		hrPrev	:	HRESULT;	(* HRESULT indicating the result of previous operations (If SUCCEEDED(hrPrev) equals false, no operation is executed.) *)
	END_VAR

END_FUNCTION

// Functions/Basic Image Operations/F_VN_ExportImageAsBmpSize

	{attribute 'TcIecLibraryType'}
	{attribute 'external_name' := 'F_VN_ExportImageAsBmpSize_GUID_8CF2EC64_9A1C_4077_EC3D_6B0E0A756AE3'}
	(* Get the required buffer size (in bytes) to store the image as bitmap. *)
	FUNCTION F_VN_ExportImageAsBmpSize : HRESULT
	VAR_INPUT
		ipImage	:	ITcVnImage;	(* Image *)
	END_VAR
	VAR_IN_OUT
		nBufferSize	:	ULINT;	(* Returns the required buffer size in bytes *)
	END_VAR
	VAR_INPUT
		hrPrev	:	HRESULT;	(* HRESULT indicating the result of previous operations (If SUCCEEDED(hrPrev) equals false, no operation is executed.) *)
	END_VAR

END_FUNCTION

// Functions/Basic Image Operations/F_VN_ExportImageAsBmpExp

	{attribute 'TcIecLibraryType'}
	{attribute 'external_name' := 'F_VN_ExportImageAsBmpExp_GUID_C458016F_97C2_4447_C5DE_B3A3BEE1F039'}
	(* Exports the image as bitmap into a given buffer (e.g. an array). F_VN_ExportImageAsBmpSizeExp should be called before to get the required buffer size. (expert function) *)
	FUNCTION F_VN_ExportImageAsBmpExp : HRESULT
	VAR_INPUT
		ipImage	:	ITcVnImage;	(* Image *)
		pBuffer	:	PVOID;	(* Pointer to a buffer to store the bitmap image (Make sure to allocate enough memory! The required size in bytes can be determined using the function F_VN_ExportImageAsBmpSizeExp) *)
		nBufferSize	:	ULINT;	(* Size of the buffer memory in bytes *)
		nWidth	:	UDINT;	(* Desired width (or 0 to keep the original width) *)
		nHeight	:	UDINT;	(* Desired height (or 0 to keep the original height) *)
		hrPrev	:	HRESULT;	(* HRESULT indicating the result of previous operations (If SUCCEEDED(hrPrev) equals false, no operation is executed.) *)
	END_VAR

END_FUNCTION

// Functions/Basic Image Operations/F_VN_ExportImageAsBmpSizeExp

	{attribute 'TcIecLibraryType'}
	{attribute 'external_name' := 'F_VN_ExportImageAsBmpSizeExp_GUID_96019CAA_540B_46D2_F9C4_B0C3FF92C8C7'}
	(* Get the required buffer size (in bytes) to store the image as bitmap. (expert function) *)
	FUNCTION F_VN_ExportImageAsBmpSizeExp : HRESULT
	VAR_INPUT
		ipImage	:	ITcVnImage;	(* Image *)
	END_VAR
	VAR_IN_OUT
		nBufferSize	:	ULINT;	(* Returns the required buffer size in bytes *)
	END_VAR
	VAR_INPUT
		nWidth	:	UDINT;	(* Desired width (or 0 to keep the original width) *)
		nHeight	:	UDINT;	(* Desired height (or 0 to keep the original height) *)
		hrPrev	:	HRESULT;	(* HRESULT indicating the result of previous operations (If SUCCEEDED(hrPrev) equals false, no operation is executed.) *)
	END_VAR

END_FUNCTION

// Functions/Basic Image Operations/F_VN_FuseImages

	{attribute 'TcIecLibraryType'}
	{attribute 'external_name' := 'F_VN_FuseImages_GUID_C7DC2A4A_D93D_43FF_E741_FF2BEC2189A5'}
	(* Fuse 2 images vertically (intended for line scan cameras). *)
	FUNCTION F_VN_FuseImages : HRESULT
	VAR_INPUT
		ipSrcImage1	:	ITcVnImage;	(* Source image 1 *)
		ipSrcImage2	:	ITcVnImage;	(* Source image 2 *)
		ipDestImage	:	REFERENCE TO ITcVnImage;	(* Destination image *)
		nFirstLine	:	UDINT;	(* Line index in ipSrcImage1, which is the first line in ipDestImage *)
		nNumLines	:	UDINT;	(* The number of lines that should be copied to ipDestImage, starting with nFirstLine in ipSrcImage1. Once the last line of ipSrcImage1 was copied, the remaining lines are copied from ipSrcImage2, starting at line index 0. *)
		hrPrev	:	HRESULT;	(* HRESULT indicating the result of previous operations (If SUCCEEDED(hrPrev) equals false, no operation is executed.) *)
	END_VAR

END_FUNCTION

// Functions/Basic Image Operations/F_VN_FuseImagesArray

	{attribute 'TcIecLibraryType'}
	{attribute 'external_name' := 'F_VN_FuseImagesArray_GUID_F3D54DA1_C1AC_44F2_E3AA_F01FD5405CEF'}
	(* Fuse up to 10 images vertically (intended for line scan cameras). *)
	FUNCTION F_VN_FuseImagesArray : HRESULT
	VAR_IN_OUT
		aSrcImageArray	:	TcVnArray10_ITcVnImage;	(* Ten-element source image array (not all elements need to be filled, nValidImages specifies the actual amount of images) *)
	END_VAR
	VAR_INPUT
		nValidImages	:	UDINT;	(* Number of valid images in aSrcImageArray *)
		ipDestImage	:	REFERENCE TO ITcVnImage;	(* Destination image *)
		nFirstLine	:	UDINT;	(* Line index in ipSrcImage1, which is the first line in ipDestImage *)
		nNumLines	:	UDINT;	(* The number of lines that should be copied to ipDestImage, starting with nFirstLine in aSrcImageArray[0]. Once the last line of aSrcImageArray[0] was copied, the remaining lines are copied from aSrcImageArray[1] (starting at line index 0) and so on. *)
		hrPrev	:	HRESULT;	(* HRESULT indicating the result of previous operations (If SUCCEEDED(hrPrev) equals false, no operation is executed.) *)
	END_VAR

END_FUNCTION

// Functions/Basic Image Operations/F_VN_GetImageChannel

	{attribute 'TcIecLibraryType'}
	{attribute 'external_name' := 'F_VN_GetImageChannel_GUID_96323F5D_F9A7_4074_DE3D_4A0975A8E41C'}
	(* Return the specified source image channel as a single-channel image. *)
	FUNCTION F_VN_GetImageChannel : HRESULT
	VAR_INPUT
		ipSrcImage	:	ITcVnImage;	(* Source image *)
		ipDestImage	:	REFERENCE TO ITcVnImage;	(* Destination image (An appropriate image will be created if required.) *)
		nChannelIndex	:	UINT;	(* Index of the requested source image channel *)
		hrPrev	:	HRESULT;	(* HRESULT indicating the result of previous operations (If SUCCEEDED(hrPrev) equals false, no operation is executed.) *)
	END_VAR

END_FUNCTION

// Functions/Basic Image Operations/F_VN_GetImageHeight

	{attribute 'TcIecLibraryType'}
	{attribute 'external_name' := 'F_VN_GetImageHeight_GUID_E6F4FF1C_FE8D_431C_D07E_8A25F97A9D44'}
	(* Return the height of an image. (Alternatively use interface method .GetHeight.) *)
	FUNCTION F_VN_GetImageHeight : HRESULT
	VAR_INPUT
		ipImage	:	ITcVnImage;	(* Image *)
	END_VAR
	VAR_IN_OUT
		nHeight	:	UDINT;	(* Return the height of ipImage *)
	END_VAR
	VAR_INPUT
		hrPrev	:	HRESULT;	(* HRESULT indicating the result of previous operations (If SUCCEEDED(hrPrev) equals false, no operation is executed.) *)
	END_VAR

END_FUNCTION

// Functions/Basic Image Operations/F_VN_GetImageInfo

	{attribute 'TcIecLibraryType'}
	{attribute 'external_name' := 'F_VN_GetImageInfo_GUID_A7B9710A_BAE9_4490_C190_B06C4F044037'}
	(* Gets a struct containing all common meta infos of the image. (Alternatively use interface method .GetImageInfo.) *)
	FUNCTION F_VN_GetImageInfo : HRESULT
	VAR_INPUT
		ipImage	:	ITcVnImage;	(* Image *)
	END_VAR
	VAR_IN_OUT
		stImageInfo	:	TcVnImageInfo;	(* Returns a struct describing the image *)
	END_VAR
	VAR_INPUT
		hrPrev	:	HRESULT;	(* HRESULT indicating the result of previous operations (If SUCCEEDED(hrPrev) equals false, no operation is executed.) *)
	END_VAR

END_FUNCTION

// Functions/Basic Image Operations/F_VN_GetImageWidth

	{attribute 'TcIecLibraryType'}
	{attribute 'external_name' := 'F_VN_GetImageWidth_GUID_DE16037B_CBBF_4F1A_CCAA_114A79EA06AE'}
	(* Return the width of an image. (Alternatively use interface method .GetWidth.) *)
	FUNCTION F_VN_GetImageWidth : HRESULT
	VAR_INPUT
		ipImage	:	ITcVnImage;	(* Image *)
	END_VAR
	VAR_IN_OUT
		nWidth	:	UDINT;	(* Return the width of ipImage *)
	END_VAR
	VAR_INPUT
		hrPrev	:	HRESULT;	(* HRESULT indicating the result of previous operations (If SUCCEEDED(hrPrev) equals false, no operation is executed.) *)
	END_VAR

END_FUNCTION

// Functions/Basic Image Operations/F_VN_GetLayoutInfo

	{attribute 'TcIecLibraryType'}
	{attribute 'external_name' := 'F_VN_GetLayoutInfo_GUID_517DAAC9_7DB1_40A4_F4A2_7CFEC75D1E68'}
	(* Return the layout information of an image *)
	FUNCTION F_VN_GetLayoutInfo : HRESULT
	VAR_INPUT
		ipImage	:	ITcVnImage;	(* Source image *)
	END_VAR
	VAR_IN_OUT
		aLayoutInfo	:	TcVnArray33_UDINT;	(* Contains layout information of ipImage. First entry of the aLayoutInfo is the number of dimensions of ipImage (max. 32), followed by the sizes of each dimension. *)
	END_VAR
	VAR_INPUT
		hrPrev	:	HRESULT;	(* HRESULT indicating the result of previous operations (If SUCCEEDED(hrPrev) equals false, no operation is executed.) *)
	END_VAR

END_FUNCTION

// Functions/Basic Image Operations/F_VN_GetPixel

	{attribute 'TcIecLibraryType'}
	{attribute 'external_name' := 'F_VN_GetPixel_GUID_DCFF0F43_C5EE_457A_DBF3_AAA75EE2168B'}
	(* Gets a specific pixel. *)
	FUNCTION F_VN_GetPixel : HRESULT
	VAR_INPUT
		ipSrcImage	:	ITcVnImage;	(* Source image *)
	END_VAR
	VAR_IN_OUT
		aValue	:	TcVnVector4_LREAL;	(* Returns the pixel value (Unused channels are set to 0.) *)
	END_VAR
	VAR_INPUT
		nX	:	UDINT;	(* x coordinate of the pixel *)
		nY	:	UDINT;	(* y coordinate of the pixel *)
		hrPrev	:	HRESULT;	(* HRESULT indicating the result of previous operations (If SUCCEEDED(hrPrev) equals false, no operation is executed.) *)
	END_VAR

END_FUNCTION

// Functions/Basic Image Operations/F_VN_GetPixelFormat

	{attribute 'TcIecLibraryType'}
	{attribute 'external_name' := 'F_VN_GetPixelFormat_GUID_57F70AB5_E99B_4292_E3FB_40AE83AF3008'}
	(* Gets the pixel format of an image. (Alternatively use interface method .GetPixelFormat.) *)
	FUNCTION F_VN_GetPixelFormat : HRESULT
	VAR_INPUT
		ipImage	:	ITcVnImage;	(* Image *)
	END_VAR
	VAR_IN_OUT
		stPixelFormat	:	TcVnPixelFormat;	(* Returns a struct describing the pixel format *)
	END_VAR
	VAR_INPUT
		hrPrev	:	HRESULT;	(* HRESULT indicating the result of previous operations (If SUCCEEDED(hrPrev) equals false, no operation is executed.) *)
	END_VAR

END_FUNCTION

// Functions/Basic Image Operations/F_VN_GetRoi

	{attribute 'TcIecLibraryType'}
	{attribute 'external_name' := 'F_VN_GetRoi_GUID_94539F10_430E_4695_D881_C8FF87B5ED42'}
	(* Gets the coordinates of the region of interest (ROI) within the image. *)
	FUNCTION F_VN_GetRoi : HRESULT
	VAR_INPUT
		ipSrcImage	:	ITcVnImage;	(* Source image *)
	END_VAR
	VAR_IN_OUT
		stRoi	:	TcVnRectangle_UDINT;	(* Returns the coordinates of the region of interest *)
	END_VAR
	VAR_INPUT
		hrPrev	:	HRESULT;	(* HRESULT indicating the result of previous operations (If SUCCEEDED(hrPrev) equals false, no operation is executed.) *)
	END_VAR

END_FUNCTION

// Functions/Basic Image Operations/F_VN_MixImageChannels

	{attribute 'TcIecLibraryType'}
	{attribute 'external_name' := 'F_VN_MixImageChannels_GUID_92D33894_7CF3_4C85_FA9E_452CA67BFF70'}
	(* Mix image channels by copying the specified channels of the source image into the specified channels of the destination image. *)
	FUNCTION F_VN_MixImageChannels : HRESULT
	VAR_INPUT
		ipSrcImage	:	ITcVnImage;	(* Source image *)
		ipDestImage	:	REFERENCE TO ITcVnImage;	(* Destination image (An appropriate image will be created if required.) *)
		ipIndicesFromTo	:	ITcVnContainer;	(* Index pairs (ContainerType_Vector_TcVnVector2_DINT), specifying which source channel (TcVnVector2_DINT [0]) should be copied to which destination channel (TcVnVector2_DINT [1]). *)
		hrPrev	:	HRESULT;	(* HRESULT indicating the result of previous operations (If SUCCEEDED(hrPrev) equals false, no operation is executed.) *)
	END_VAR

END_FUNCTION

// Functions/Basic Image Operations/F_VN_ResetRoi

	{attribute 'TcIecLibraryType'}
	{attribute 'external_name' := 'F_VN_ResetRoi_GUID_44C3AC67_64D8_4846_C571_84F70E9C0041'}
	(* Reset the region of interest (ROI) of an image. (After this operation, the ROI is set to the entire image.) *)
	FUNCTION F_VN_ResetRoi : HRESULT
	VAR_INPUT
		ipImage	:	ITcVnImage;	(* Image *)
		hrPrev	:	HRESULT;	(* HRESULT indicating the result of previous operations (If SUCCEEDED(hrPrev) equals false, no operation is executed.) *)
	END_VAR

END_FUNCTION

// Functions/Basic Image Operations/F_VN_SetImageChannel

	{attribute 'TcIecLibraryType'}
	{attribute 'external_name' := 'F_VN_SetImageChannel_GUID_6282859E_3953_4166_ED00_BDBEA2E5C044'}
	(* Sets the specified destination image channel to the values of the specified source image channel. *)
	FUNCTION F_VN_SetImageChannel : HRESULT
	VAR_INPUT
		ipSrcImage	:	ITcVnImage;	(* Source image *)
		ipDestImage	:	REFERENCE TO ITcVnImage;	(* Destination image (An appropriate image will be created if required.) *)
		nSrcChannelIndex	:	UINT;	(* Index of the source image channel *)
		nDestChannelIndex	:	UINT;	(* Index of the destination image channel, which will be replaced by the specified source image channel *)
		hrPrev	:	HRESULT;	(* HRESULT indicating the result of previous operations (If SUCCEEDED(hrPrev) equals false, no operation is executed.) *)
	END_VAR

END_FUNCTION

// Functions/Basic Image Operations/F_VN_SetPixel

	{attribute 'TcIecLibraryType'}
	{attribute 'external_name' := 'F_VN_SetPixel_GUID_E3D7AD87_631F_453C_CA06_16FFFAAED977'}
	(* Sets a specific pixel. *)
	FUNCTION F_VN_SetPixel : HRESULT
	VAR_INPUT
		ipSrcImage	:	ITcVnImage;	(* Source image *)
	END_VAR
	VAR_IN_OUT
		aValue	:	TcVnVector4_LREAL;	(* The pixel value to set (additional channels are ignored.) *)
	END_VAR
	VAR_INPUT
		nX	:	UDINT;	(* x coordinate of the pixel *)
		nY	:	UDINT;	(* y coordinate of the pixel *)
		hrPrev	:	HRESULT;	(* HRESULT indicating the result of previous operations (If SUCCEEDED(hrPrev) equals false, no operation is executed.) *)
	END_VAR

END_FUNCTION

// Functions/Basic Image Operations/F_VN_SetPixels

	{attribute 'TcIecLibraryType'}
	{attribute 'external_name' := 'F_VN_SetPixels_GUID_92708F63_07CE_4BF8_CCED_0CA1DBADF248'}
	(* Sets all pixels of an image to a given value. *)
	FUNCTION F_VN_SetPixels : HRESULT
	VAR_INPUT
		ipDestImage	:	ITcVnImage;	(* Destination image *)
	END_VAR
	VAR_IN_OUT
		aValue	:	TcVnVector4_LREAL;	(* Pixel value *)
	END_VAR
	VAR_INPUT
		hrPrev	:	HRESULT;	(* HRESULT indicating the result of previous operations (If SUCCEEDED(hrPrev) equals false, no operation is executed.) *)
	END_VAR

END_FUNCTION

// Functions/Basic Image Operations/F_VN_SetPixelsExp

	{attribute 'TcIecLibraryType'}
	{attribute 'external_name' := 'F_VN_SetPixelsExp_GUID_2D58912C_21E3_4754_D874_F9B91D2F57D2'}
	(* Sets all pixels of an image to a given value. (expert function) *)
	FUNCTION F_VN_SetPixelsExp : HRESULT
	VAR_INPUT
		ipDestImage	:	ITcVnImage;	(* Destination image *)
	END_VAR
	VAR_IN_OUT
		aValue	:	TcVnVector4_LREAL;	(* Pixel value *)
	END_VAR
	VAR_INPUT
		ipMask	:	ITcVnImage;	(* Mask image *)
		hrPrev	:	HRESULT;	(* HRESULT indicating the result of previous operations (If SUCCEEDED(hrPrev) equals false, no operation is executed.) *)
	END_VAR

END_FUNCTION

// Functions/Basic Image Operations/F_VN_SetRoi

	{attribute 'TcIecLibraryType'}
	{attribute 'external_name' := 'F_VN_SetRoi_GUID_03CC3B69_B131_4127_D0E9_3F642AB7AA72'}
	(* Sets a region of interest (ROI) within an image. *)
	FUNCTION F_VN_SetRoi : HRESULT
	VAR_INPUT
		nX	:	UDINT;	(* Left boundary (inclusive 0-based index) *)
		nY	:	UDINT;	(* Upper boundary (inclusive 0-based index) *)
		nWidth	:	UDINT;	(* ROI width *)
		nHeight	:	UDINT;	(* ROI height *)
		ipDestImage	:	ITcVnImage;	(* Destination image *)
		hrPrev	:	HRESULT;	(* HRESULT indicating the result of previous operations (If SUCCEEDED(hrPrev) equals false, no operation is executed.) *)
	END_VAR

END_FUNCTION

// Functions/Basic Image Operations/F_VN_SetRoi_TcVnRectangle_DINT

	{attribute 'TcIecLibraryType'}
	{attribute 'external_name' := 'F_VN_SetRoi_TcVnRectangle_DINT_GUID_5D877643_EF8D_47ED_C9B7_C78D1649D2D1'}
	(* Sets a region of interest (ROI) within an image. *)
	FUNCTION F_VN_SetRoi_TcVnRectangle_DINT : HRESULT
	VAR_IN_OUT
		stRoi	:	TcVnRectangle_DINT;	(* Region of interest *)
	END_VAR
	VAR_INPUT
		ipDestImage	:	ITcVnImage;	(* Destination image *)
		hrPrev	:	HRESULT;	(* HRESULT indicating the result of previous operations (If SUCCEEDED(hrPrev) equals false, no operation is executed.) *)
	END_VAR

END_FUNCTION

// Functions/Basic Image Operations/F_VN_SetRoi_TcVnRectangle_UDINT

	{attribute 'TcIecLibraryType'}
	{attribute 'external_name' := 'F_VN_SetRoi_TcVnRectangle_UDINT_GUID_08BD351B_44D9_4D5C_CE14_16CF5906D143'}
	(* Sets a region of interest (ROI) within an image. *)
	FUNCTION F_VN_SetRoi_TcVnRectangle_UDINT : HRESULT
	VAR_IN_OUT
		stRoi	:	TcVnRectangle_UDINT;	(* Region of interest *)
	END_VAR
	VAR_INPUT
		ipDestImage	:	ITcVnImage;	(* Destination image *)
		hrPrev	:	HRESULT;	(* HRESULT indicating the result of previous operations (If SUCCEEDED(hrPrev) equals false, no operation is executed.) *)
	END_VAR

END_FUNCTION

// Functions/Basic Image Operations/F_VN_SplitImageChannels

	{attribute 'TcIecLibraryType'}
	{attribute 'external_name' := 'F_VN_SplitImageChannels_GUID_C1CD0E12_94A9_4EC9_DC81_980A69742BBB'}
	(* Split a multi-channel image into multiple single channel images (1 for each source image channel). *)
	FUNCTION F_VN_SplitImageChannels : HRESULT
	VAR_INPUT
		ipSrcImage	:	ITcVnImage;	(* Source image with multiple channels *)
		pDestImages	:	PVOID;	(* Pointer to an array of ITcVnImage (appropriate destination images will be created if required) *)
		nArraySize	:	UINT;	(* Number of pDestImages array elements (array must be >= ipSourceImage channels) *)
		hrPrev	:	HRESULT;	(* HRESULT indicating the result of previous operations (If SUCCEEDED(hrPrev) equals false, no operation is executed.) *)
	END_VAR
	VAR_OUTPUT
		nImageChannels	:	UINT;	(* Actual source image channels *)
	END_VAR

END_FUNCTION

// Functions/Basic Image Operations/F_VN_TransformIntoDisplayableImageExp

	{attribute 'TcIecLibraryType'}
	{attribute 'external_name' := 'F_VN_TransformIntoDisplayableImageExp_GUID_7EE9CC3A_7888_45A0_D6B5_29E01D0A57CC'}
	(* Transform an image into a displayable image. The source image will be released and zeroed while existing destination images will be released and overwritten with the function result. If bAllowDeepCopy equals false, the source image must not be used anywhere else and the transformation is always very fast. Otherwise, if bAllowDeepCopy equals true, a deep copy of the source image might be created if required, which will result in a longer execution time. If you want to use ipSrcImage after this function call, use F_VN_CopyIntoDisplayableImage instead. (expert function) *)
	FUNCTION F_VN_TransformIntoDisplayableImageExp : HRESULT
	VAR_INPUT
		ipSrcImage	:	REFERENCE TO ITcVnImage;	(* Source image *)
		ipDestImage	:	REFERENCE TO ITcVnDisplayableImage;	(* Returns the displayable image *)
		bAllowDeepCopy	:	BOOL;	(* Allow deep image copies, if required *)
		hrPrev	:	HRESULT;	(* HRESULT indicating the result of previous operations (If SUCCEEDED(hrPrev) equals false, no operation is executed.) *)
	END_VAR

END_FUNCTION

// Functions/Container Statistics/F_VN_ContainerAverage

	{attribute 'TcIecLibraryType'}
	{attribute 'external_name' := 'F_VN_ContainerAverage_GUID_C21B6E9C_FC5B_45AB_FDF2_7C6B9C752351'}
	(* Calculate the average of elements in a container. *)
	FUNCTION F_VN_ContainerAverage : HRESULT
	VAR_INPUT
		ipSrcContainer	:	ITcVnContainer;	(* Source container (Arithmetic, point and vector element types are supported. For points and vectors, the euclidean norm is used.) *)
	END_VAR
	VAR_IN_OUT
		fAverage	:	LREAL;	(* Returns the calculated average value *)
	END_VAR
	VAR_INPUT
		hrPrev	:	HRESULT;	(* HRESULT indicating the result of previous operations (If SUCCEEDED(hrPrev) equals false, no operation is executed.) *)
	END_VAR

END_FUNCTION

// Functions/Container Statistics/F_VN_ContainerAverageElementwise2

	{attribute 'TcIecLibraryType'}
	{attribute 'external_name' := 'F_VN_ContainerAverageElementwise2_GUID_CD05DEC3_2CC2_475C_F448_F85D940E8B13'}
	(* Calculate the elementwise average of 2D elements in a container. *)
	FUNCTION F_VN_ContainerAverageElementwise2 : HRESULT
	VAR_INPUT
		ipSrcContainer	:	ITcVnContainer;	(* Source container with 2D points or vectors *)
	END_VAR
	VAR_IN_OUT
		aAverage	:	TcVnVector2_LREAL;	(* Returns the calculated average values *)
	END_VAR
	VAR_INPUT
		hrPrev	:	HRESULT;	(* HRESULT indicating the result of previous operations (If SUCCEEDED(hrPrev) equals false, no operation is executed.) *)
	END_VAR

END_FUNCTION

// Functions/Container Statistics/F_VN_ContainerAverageElementwise3

	{attribute 'TcIecLibraryType'}
	{attribute 'external_name' := 'F_VN_ContainerAverageElementwise3_GUID_286D05ED_21BB_4D0D_D161_A9A600960F71'}
	(* Calculate the elementwise average of 3D elements in a container. *)
	FUNCTION F_VN_ContainerAverageElementwise3 : HRESULT
	VAR_INPUT
		ipSrcContainer	:	ITcVnContainer;	(* Source container with 3D points or vectors *)
	END_VAR
	VAR_IN_OUT
		aAverage	:	TcVnVector3_LREAL;	(* Returns the calculated average values *)
	END_VAR
	VAR_INPUT
		hrPrev	:	HRESULT;	(* HRESULT indicating the result of previous operations (If SUCCEEDED(hrPrev) equals false, no operation is executed.) *)
	END_VAR

END_FUNCTION

// Functions/Container Statistics/F_VN_ContainerAverageElementwise4

	{attribute 'TcIecLibraryType'}
	{attribute 'external_name' := 'F_VN_ContainerAverageElementwise4_GUID_B63FAAD7_930A_44F9_F8FC_0007B2A07E13'}
	(* Calculate the elementwise average of 4D elements in a container. *)
	FUNCTION F_VN_ContainerAverageElementwise4 : HRESULT
	VAR_INPUT
		ipSrcContainer	:	ITcVnContainer;	(* Source container with 4D vectors *)
	END_VAR
	VAR_IN_OUT
		aAverage	:	TcVnVector4_LREAL;	(* Returns the calculated average values *)
	END_VAR
	VAR_INPUT
		hrPrev	:	HRESULT;	(* HRESULT indicating the result of previous operations (If SUCCEEDED(hrPrev) equals false, no operation is executed.) *)
	END_VAR

END_FUNCTION

// Functions/Container Statistics/F_VN_ContainerAverageVariance

	{attribute 'TcIecLibraryType'}
	{attribute 'external_name' := 'F_VN_ContainerAverageVariance_GUID_90FE02D6_6CC1_49D5_F306_DDD9A1425DF1'}
	(* Calculate the average and variance of elements in a container. *)
	FUNCTION F_VN_ContainerAverageVariance : HRESULT
	VAR_INPUT
		ipSrcContainer	:	ITcVnContainer;	(* Source container (Arithmetic, point and vector element types are supported. For points and vectors, the euclidean norm is used.) *)
	END_VAR
	VAR_IN_OUT
		fAverage	:	LREAL;	(* Returns the calculated average value *)
		fVariance	:	LREAL;	(* Returns the calculated variance value *)
	END_VAR
	VAR_INPUT
		hrPrev	:	HRESULT;	(* HRESULT indicating the result of previous operations (If SUCCEEDED(hrPrev) equals false, no operation is executed.) *)
	END_VAR

END_FUNCTION

// Functions/Container Statistics/F_VN_ContainerAverageVarianceElementwise2

	{attribute 'TcIecLibraryType'}
	{attribute 'external_name' := 'F_VN_ContainerAverageVarianceElementwise2_GUID_F54B809D_B72F_4220_FE5A_A0887EB15428'}
	(* Calculate the elementwise average and variance of 2D elements in a container. *)
	FUNCTION F_VN_ContainerAverageVarianceElementwise2 : HRESULT
	VAR_INPUT
		ipSrcContainer	:	ITcVnContainer;	(* Source container with 2D points or vectors *)
	END_VAR
	VAR_IN_OUT
		aAverage	:	TcVnVector2_LREAL;	(* Returns the calculated average values *)
		aVariance	:	TcVnVector2_LREAL;	(* Returns the calculated variance values *)
	END_VAR
	VAR_INPUT
		hrPrev	:	HRESULT;	(* HRESULT indicating the result of previous operations (If SUCCEEDED(hrPrev) equals false, no operation is executed.) *)
	END_VAR

END_FUNCTION

// Functions/Container Statistics/F_VN_ContainerAverageVarianceElementwise3

	{attribute 'TcIecLibraryType'}
	{attribute 'external_name' := 'F_VN_ContainerAverageVarianceElementwise3_GUID_92100E32_075B_4ACD_EBC6_6D0E2E61BB14'}
	(* Calculate the elementwise average and variance of 3D elements in a container. *)
	FUNCTION F_VN_ContainerAverageVarianceElementwise3 : HRESULT
	VAR_INPUT
		ipSrcContainer	:	ITcVnContainer;	(* Source container with 3D points or vectors *)
	END_VAR
	VAR_IN_OUT
		aAverage	:	TcVnVector3_LREAL;	(* Returns the calculated average values *)
		aVariance	:	TcVnVector3_LREAL;	(* Returns the calculated variance values *)
	END_VAR
	VAR_INPUT
		hrPrev	:	HRESULT;	(* HRESULT indicating the result of previous operations (If SUCCEEDED(hrPrev) equals false, no operation is executed.) *)
	END_VAR

END_FUNCTION

// Functions/Container Statistics/F_VN_ContainerAverageVarianceElementwise4

	{attribute 'TcIecLibraryType'}
	{attribute 'external_name' := 'F_VN_ContainerAverageVarianceElementwise4_GUID_6B8D4DAE_B53E_4414_C27E_3C7F1BC1A558'}
	(* Calculate the elementwise average and variance of 4D elements in a container. *)
	FUNCTION F_VN_ContainerAverageVarianceElementwise4 : HRESULT
	VAR_INPUT
		ipSrcContainer	:	ITcVnContainer;	(* Source container with 4D vectors *)
	END_VAR
	VAR_IN_OUT
		aAverage	:	TcVnVector4_LREAL;	(* Returns the calculated average values *)
		aVariance	:	TcVnVector4_LREAL;	(* Returns the calculated variance values *)
	END_VAR
	VAR_INPUT
		hrPrev	:	HRESULT;	(* HRESULT indicating the result of previous operations (If SUCCEEDED(hrPrev) equals false, no operation is executed.) *)
	END_VAR

END_FUNCTION

// Functions/Container Statistics/F_VN_MaxElement

	{attribute 'TcIecLibraryType'}
	{attribute 'external_name' := 'F_VN_MaxElement_GUID_FBC0ECFD_EEC1_4B36_D212_017BCDA8DA46'}
	(* Gets the maximum element of a container. *)
	FUNCTION F_VN_MaxElement : HRESULT
	VAR_INPUT
		ipSrcContainer	:	ITcVnContainer;	(* Source container (Arithmetic, point and vector element types are supported. For points and vectors, the euclidean norm is used.) *)
		ipDestIterator	:	REFERENCE TO ITcVnBidirectionalIterator;	(* Returns an iterator to the requested element *)
	END_VAR
	VAR_IN_OUT
		nIndex	:	ULINT;	(* Returns the position of the requested element within the container *)
	END_VAR
	VAR_INPUT
		hrPrev	:	HRESULT;	(* HRESULT indicating the result of previous operations (If SUCCEEDED(hrPrev) equals false, no operation is executed.) *)
	END_VAR

END_FUNCTION

// Functions/Container Statistics/F_VN_MedianElement

	{attribute 'TcIecLibraryType'}
	{attribute 'external_name' := 'F_VN_MedianElement_GUID_1BD5537E_FA80_4573_C96F_A1EE778BF94F'}
	(* Gets the median element of a container. *)
	FUNCTION F_VN_MedianElement : HRESULT
	VAR_INPUT
		ipSrcContainer	:	ITcVnContainer;	(* Source container (Arithmetic, point and vector element types are supported. For points and vectors, the euclidean norm is used.) *)
		ipDestIterator	:	REFERENCE TO ITcVnBidirectionalIterator;	(* Returns an iterator to the requested element *)
	END_VAR
	VAR_IN_OUT
		nIndex	:	ULINT;	(* Returns the position of the requested element within the container *)
	END_VAR
	VAR_INPUT
		hrPrev	:	HRESULT;	(* HRESULT indicating the result of previous operations (If SUCCEEDED(hrPrev) equals false, no operation is executed.) *)
	END_VAR

END_FUNCTION

// Functions/Container Statistics/F_VN_MinElement

	{attribute 'TcIecLibraryType'}
	{attribute 'external_name' := 'F_VN_MinElement_GUID_FDF0B19D_EAEC_4906_F620_AD7F87BACC68'}
	(* Gets the minimum element of a container. *)
	FUNCTION F_VN_MinElement : HRESULT
	VAR_INPUT
		ipSrcContainer	:	ITcVnContainer;	(* Source container (Arithmetic, point and vector element types are supported. For points and vectors, the euclidean norm is used.) *)
		ipDestIterator	:	REFERENCE TO ITcVnBidirectionalIterator;	(* Returns an iterator to the requested element *)
	END_VAR
	VAR_IN_OUT
		nIndex	:	ULINT;	(* Returns the position of the requested element within the container *)
	END_VAR
	VAR_INPUT
		hrPrev	:	HRESULT;	(* HRESULT indicating the result of previous operations (If SUCCEEDED(hrPrev) equals false, no operation is executed.) *)
	END_VAR

END_FUNCTION

// Functions/Fourier Analysis/F_VN_CreateBandpassButterworthFilter

	{attribute 'TcIecLibraryType'}
	{attribute 'external_name' := 'F_VN_CreateBandpassButterworthFilter_GUID_CCE2CE6D_57D0_48A7_F403_8D142F6A2BC0'}
	(* Creates a bandpass Butterworth filter, which can be applied to a frequency domain image by element-wise multiplication. *)
	FUNCTION F_VN_CreateBandpassButterworthFilter : HRESULT
	VAR_INPUT
		ipFilter	:	REFERENCE TO ITcVnImage;	(* Returns the created filter (1 channel of type REAL or LREAL, depending on bDoublePrecision. Non-zero interface pointers are reused.). *)
		nWidth	:	UDINT;	(* Filter width (even, >= 2, must match the width of the image it is applied to) *)
		nHeight	:	UDINT;	(* Filter height (even, >= 2, must match the height of the image it is applied to) *)
		bDoublePrecision	:	BOOL;	(* If true, the filter is generated with double precision (LREAL) instead of single precision (REAL). *)
		bOriginAtCenter	:	BOOL;	(* If true, the filter origin is shifted to the image center. *)
		fCutoffDistance	:	LREAL;	(* The cutoff distance of the Butterworth filter (> 0). *)
		fBandWidth	:	LREAL;	(* The band width of the Butterworth filter (> 0). *)
		nOrder	:	UDINT;	(* The order of the Butterworth filter (> 0). *)
		fScale	:	LREAL;	(* The scale factor of the Butterworth filter denominator term (> 0, e.g. 0.414 or 1.0). *)
		hrPrev	:	HRESULT;	(* HRESULT indicating the result of previous operations (If SUCCEEDED(hrPrev) equals false, no operation is executed.) *)
	END_VAR

END_FUNCTION

// Functions/Fourier Analysis/F_VN_CreateBandpassGaussianFilter

	{attribute 'TcIecLibraryType'}
	{attribute 'external_name' := 'F_VN_CreateBandpassGaussianFilter_GUID_C3AD5AA0_6523_4BD9_C6D1_9B7DF138EC3F'}
	(* Creates a bandpass Gaussian filter, which can be applied to a frequency domain image by element-wise multiplication. *)
	FUNCTION F_VN_CreateBandpassGaussianFilter : HRESULT
	VAR_INPUT
		ipFilter	:	REFERENCE TO ITcVnImage;	(* Returns the created filter (1 channel of type REAL or LREAL, depending on bDoublePrecision. Non-zero interface pointers are reused.). *)
		nWidth	:	UDINT;	(* Filter width (even, >= 2, must match the width of the image it is applied to) *)
		nHeight	:	UDINT;	(* Filter height (even, >= 2, must match the height of the image it is applied to) *)
		bDoublePrecision	:	BOOL;	(* If true, the filter is generated with double precision (LREAL) instead of single precision (REAL). *)
		bOriginAtCenter	:	BOOL;	(* If true, the filter origin is shifted to the image center. *)
		fCutoffDistance	:	LREAL;	(* The cutoff distance of the Gaussian filter (> 0). *)
		fBandWidth	:	LREAL;	(* The band width of the Gaussian filter (> 0). *)
		hrPrev	:	HRESULT;	(* HRESULT indicating the result of previous operations (If SUCCEEDED(hrPrev) equals false, no operation is executed.) *)
	END_VAR

END_FUNCTION

// Functions/Fourier Analysis/F_VN_CreateBandrejectButterworthFilter

	{attribute 'TcIecLibraryType'}
	{attribute 'external_name' := 'F_VN_CreateBandrejectButterworthFilter_GUID_2B6E5925_FDAB_4940_D8CB_101A95241A81'}
	(* Creates a bandreject Butterworth filter, which can be applied to a frequency domain image by element-wise multiplication. *)
	FUNCTION F_VN_CreateBandrejectButterworthFilter : HRESULT
	VAR_INPUT
		ipFilter	:	REFERENCE TO ITcVnImage;	(* Returns the created filter (1 channel of type REAL or LREAL, depending on bDoublePrecision. Non-zero interface pointers are reused.). *)
		nWidth	:	UDINT;	(* Filter width (even, >= 2, must match the width of the image it is applied to) *)
		nHeight	:	UDINT;	(* Filter height (even, >= 2, must match the height of the image it is applied to) *)
		bDoublePrecision	:	BOOL;	(* If true, the filter is generated with double precision (LREAL) instead of single precision (REAL). *)
		bOriginAtCenter	:	BOOL;	(* If true, the filter origin is shifted to the image center. *)
		fCutoffDistance	:	LREAL;	(* The cutoff distance of the Butterworth filter (> 0). *)
		fBandWidth	:	LREAL;	(* The band width of the Butterworth filter (> 0). *)
		nOrder	:	UDINT;	(* The order of the Butterworth filter (> 0). *)
		fScale	:	LREAL;	(* The scale factor of the Butterworth filter denominator term (> 0, e.g. 0.414 or 1.0). *)
		hrPrev	:	HRESULT;	(* HRESULT indicating the result of previous operations (If SUCCEEDED(hrPrev) equals false, no operation is executed.) *)
	END_VAR

END_FUNCTION

// Functions/Fourier Analysis/F_VN_CreateBandrejectGaussianFilter

	{attribute 'TcIecLibraryType'}
	{attribute 'external_name' := 'F_VN_CreateBandrejectGaussianFilter_GUID_45905B62_0316_4B70_C8A9_559F3D0A7C42'}
	(* Creates a bandreject Gaussian filter, which can be applied to a frequency domain image by element-wise multiplication. *)
	FUNCTION F_VN_CreateBandrejectGaussianFilter : HRESULT
	VAR_INPUT
		ipFilter	:	REFERENCE TO ITcVnImage;	(* Returns the created filter (1 channel of type REAL or LREAL, depending on bDoublePrecision. Non-zero interface pointers are reused.). *)
		nWidth	:	UDINT;	(* Filter width (even, >= 2, must match the width of the image it is applied to) *)
		nHeight	:	UDINT;	(* Filter height (even, >= 2, must match the height of the image it is applied to) *)
		bDoublePrecision	:	BOOL;	(* If true, the filter is generated with double precision (LREAL) instead of single precision (REAL). *)
		bOriginAtCenter	:	BOOL;	(* If true, the filter origin is shifted to the image center. *)
		fCutoffDistance	:	LREAL;	(* The cutoff distance of the Gaussian filter (> 0). *)
		fBandWidth	:	LREAL;	(* The band width of the Gaussian filter (> 0). *)
		hrPrev	:	HRESULT;	(* HRESULT indicating the result of previous operations (If SUCCEEDED(hrPrev) equals false, no operation is executed.) *)
	END_VAR

END_FUNCTION

// Functions/Fourier Analysis/F_VN_CreateHighpassButterworthFilter

	{attribute 'TcIecLibraryType'}
	{attribute 'external_name' := 'F_VN_CreateHighpassButterworthFilter_GUID_4EA20F58_03AF_4524_DF35_FDC161A94F29'}
	(* Creates a highpass Butterworth filter, which can be applied to a frequency domain image by element-wise multiplication. *)
	FUNCTION F_VN_CreateHighpassButterworthFilter : HRESULT
	VAR_INPUT
		ipFilter	:	REFERENCE TO ITcVnImage;	(* Returns the created filter (1 channel of type REAL or LREAL, depending on bDoublePrecision. Non-zero interface pointers are reused.). *)
		nWidth	:	UDINT;	(* Filter width (even, >= 2, must match the width of the image it is applied to) *)
		nHeight	:	UDINT;	(* Filter height (even, >= 2, must match the height of the image it is applied to) *)
		bDoublePrecision	:	BOOL;	(* If true, the filter is generated with double precision (LREAL) instead of single precision (REAL). *)
		bOriginAtCenter	:	BOOL;	(* If true, the filter origin is shifted to the image center. *)
		fCutoffDistance	:	LREAL;	(* The cutoff distance of the Butterworth filter (> 0). *)
		nOrder	:	UDINT;	(* The order of the Butterworth filter (> 0). *)
		fScale	:	LREAL;	(* The scale factor of the Butterworth filter denominator term (> 0, e.g. 0.414 or 1.0). *)
		hrPrev	:	HRESULT;	(* HRESULT indicating the result of previous operations (If SUCCEEDED(hrPrev) equals false, no operation is executed.) *)
	END_VAR

END_FUNCTION

// Functions/Fourier Analysis/F_VN_CreateHighpassGaussianFilter

	{attribute 'TcIecLibraryType'}
	{attribute 'external_name' := 'F_VN_CreateHighpassGaussianFilter_GUID_F9269179_898C_4929_FE65_D9F81B8BDED8'}
	(* Creates a highpass Gaussian filter, which can be applied to a frequency domain image by element-wise multiplication. *)
	FUNCTION F_VN_CreateHighpassGaussianFilter : HRESULT
	VAR_INPUT
		ipFilter	:	REFERENCE TO ITcVnImage;	(* Returns the created filter (1 channel of type REAL or LREAL, depending on bDoublePrecision. Non-zero interface pointers are reused.). *)
		nWidth	:	UDINT;	(* Filter width (even, >= 2, must match the width of the image it is applied to) *)
		nHeight	:	UDINT;	(* Filter height (even, >= 2, must match the height of the image it is applied to) *)
		bDoublePrecision	:	BOOL;	(* If true, the filter is generated with double precision (LREAL) instead of single precision (REAL). *)
		bOriginAtCenter	:	BOOL;	(* If true, the filter origin is shifted to the image center. *)
		fCutoffDistance	:	LREAL;	(* The cutoff distance of the Gaussian filter (> 0). *)
		hrPrev	:	HRESULT;	(* HRESULT indicating the result of previous operations (If SUCCEEDED(hrPrev) equals false, no operation is executed.) *)
	END_VAR

END_FUNCTION

// Functions/Fourier Analysis/F_VN_CreateLowpassButterworthFilter

	{attribute 'TcIecLibraryType'}
	{attribute 'external_name' := 'F_VN_CreateLowpassButterworthFilter_GUID_5FA3C211_598F_4E5F_D34F_22C524ED6407'}
	(* Creates a lowpass Butterworth filter, which can be applied to a frequency domain image by element-wise multiplication. *)
	FUNCTION F_VN_CreateLowpassButterworthFilter : HRESULT
	VAR_INPUT
		ipFilter	:	REFERENCE TO ITcVnImage;	(* Returns the created filter (1 channel of type REAL or LREAL, depending on bDoublePrecision. Non-zero interface pointers are reused.). *)
		nWidth	:	UDINT;	(* Filter width (even, >= 2, must match the width of the image it is applied to) *)
		nHeight	:	UDINT;	(* Filter height (even, >= 2, must match the height of the image it is applied to) *)
		bDoublePrecision	:	BOOL;	(* If true, the filter is generated with double precision (LREAL) instead of single precision (REAL). *)
		bOriginAtCenter	:	BOOL;	(* If true, the filter origin is shifted to the image center. *)
		fCutoffDistance	:	LREAL;	(* The cutoff distance of the Butterworth filter (> 0). *)
		nOrder	:	UDINT;	(* The order of the Butterworth filter (> 0). *)
		fScale	:	LREAL;	(* The scale factor of the Butterworth filter denominator term (> 0, e.g. 0.414 or 1.0). *)
		hrPrev	:	HRESULT;	(* HRESULT indicating the result of previous operations (If SUCCEEDED(hrPrev) equals false, no operation is executed.) *)
	END_VAR

END_FUNCTION

// Functions/Fourier Analysis/F_VN_CreateLowpassGaussianFilter

	{attribute 'TcIecLibraryType'}
	{attribute 'external_name' := 'F_VN_CreateLowpassGaussianFilter_GUID_94A5082D_671A_4064_F027_C6195DFC7619'}
	(* Creates a lowpass Gaussian filter, which can be applied to a frequency domain image by element-wise multiplication. *)
	FUNCTION F_VN_CreateLowpassGaussianFilter : HRESULT
	VAR_INPUT
		ipFilter	:	REFERENCE TO ITcVnImage;	(* Returns the created filter (1 channel of type REAL or LREAL, depending on bDoublePrecision. Non-zero interface pointers are reused.). *)
		nWidth	:	UDINT;	(* Filter width (even, >= 2, must match the width of the image it is applied to) *)
		nHeight	:	UDINT;	(* Filter height (even, >= 2, must match the height of the image it is applied to) *)
		bDoublePrecision	:	BOOL;	(* If true, the filter is generated with double precision (LREAL) instead of single precision (REAL). *)
		bOriginAtCenter	:	BOOL;	(* If true, the filter origin is shifted to the image center. *)
		fCutoffDistance	:	LREAL;	(* The cutoff distance of the Gaussian filter (> 0). *)
		hrPrev	:	HRESULT;	(* HRESULT indicating the result of previous operations (If SUCCEEDED(hrPrev) equals false, no operation is executed.) *)
	END_VAR

END_FUNCTION

// Functions/Fourier Analysis/F_VN_Dft

	{attribute 'TcIecLibraryType'}
	{attribute 'external_name' := 'F_VN_Dft_GUID_F441B72F_E58C_425D_F64D_6F7161506BE6'}
	(* Computes the DFT for a given image. *)
	FUNCTION F_VN_Dft : HRESULT
	VAR_INPUT
		ipSpatialImage	:	ITcVnImage;	(* Source image (elements of type REAL or LREAL, 1 (Re) or 2 (Re + Im) channels) *)
		ipFrequencyImage	:	REFERENCE TO ITcVnImage;	(* Destination image (same type as ipSpatialImage, but number of channels and size can vary depending on bPackedCCS and bAutoPadding. *)
		bPackedCCS	:	BOOL;	(* If true and ipSpatialImage has only 1 channel, the result image will have 1 channel with packed complex-conjugate-symmetrical format results. Otherwise, the result image will have 2 separate channels (Re + Im), containing the full spectrum. *)
		bAutoPadding	:	BOOL;	(* If true, the input image is automatically padded (with 0s) to optimal size if required, to speed up dft (Creates a temporary copy so that ipSpatialImage content stays unchanged, which also requires some additional computation power. Therefore, it is recommended to compare execution times with and without padding.) *)
		hrPrev	:	HRESULT;	(* HRESULT indicating the result of previous operations (If SUCCEEDED(hrPrev) equals false, no operation is executed.) *)
	END_VAR

END_FUNCTION

// Functions/Fourier Analysis/F_VN_InverseDft

	{attribute 'TcIecLibraryType'}
	{attribute 'external_name' := 'F_VN_InverseDft_GUID_39039517_580B_43E6_D7B3_F7E5CFC4DC54'}
	(* Compute the inverse DFT for a given frequency image. *)
	FUNCTION F_VN_InverseDft : HRESULT
	VAR_INPUT
		ipFrequencyImage	:	ITcVnImage;	(* Source frequency image (elements of type REAL or LREAL, 1 (packed CCS) or 2 (Re + Im) channels) *)
		ipSpatialImage	:	REFERENCE TO ITcVnImage;	(* Destination image (Same type as ipFrequencyImage, but number of channels can vary depending on bRealOutput. An appropriate image will be created if required.) *)
		bRealOutput	:	BOOL;	(* Only relevant if ipFrequencyImage has 2 channels. If true, the result image will have only 1 channel. Otherwise, the result image will have 2 separate channels (Re + Im). If ipFrequencyImage has only 1 channel, packed CCS format is assumed and the result image will always have only 1 channel. *)
		hrPrev	:	HRESULT;	(* HRESULT indicating the result of previous operations (If SUCCEEDED(hrPrev) equals false, no operation is executed.) *)
	END_VAR

END_FUNCTION

// Functions/Fourier Analysis/F_VN_OptimalDftSize

	{attribute 'TcIecLibraryType'}
	{attribute 'external_name' := 'F_VN_OptimalDftSize_GUID_17E1FAFB_84B6_4D17_ED79_3CD0623BBE40'}
	(* Computes the optimal image size for applying a dft (can lead to better performance). *)
	FUNCTION F_VN_OptimalDftSize : HRESULT
	VAR_INPUT
		ipImage	:	ITcVnImage;	(* Source image for which to compute the optimal width and height *)
	END_VAR
	VAR_IN_OUT
		nOptWidth	:	UDINT;	(* Returns the optimal width of the image *)
		nOptHeight	:	UDINT;	(* Returns the optimal height of the image *)
	END_VAR
	VAR_INPUT
		hrPrev	:	HRESULT;	(* HRESULT indicating the result of previous operations (If SUCCEEDED(hrPrev) equals false, no operation is executed.) *)
	END_VAR

END_FUNCTION

// Functions/Fourier Analysis/F_VN_PadImageBorder

	{attribute 'TcIecLibraryType'}
	{attribute 'external_name' := 'F_VN_PadImageBorder_GUID_6A5C3322_7CFD_40CD_D198_92131E93C05F'}
	(* Add padding (zeros) around the original image borders. *)
	FUNCTION F_VN_PadImageBorder : HRESULT
	VAR_INPUT
		ipSrcImage	:	ITcVnImage;	(* Source image *)
		ipPaddedImage	:	REFERENCE TO ITcVnImage;	(* Padded destination image (Same type as ipSrcImage, an appropriate destination image will be created if required.) *)
		nTopBorder	:	UDINT;	(* Padding height in pixels above top border *)
		nBottomBorder	:	UDINT;	(* Padding height in pixels below bottom border *)
		nLeftBorder	:	UDINT;	(* Padding width in pixels before left border *)
		nRightBorder	:	UDINT;	(* Padding width in pixels after right border *)
		hrPrev	:	HRESULT;	(* HRESULT indicating the result of previous operations (If SUCCEEDED(hrPrev) equals false, no operation is executed.) *)
	END_VAR

END_FUNCTION

// Functions/Fourier Analysis/F_VN_PadImageBorderExp

	{attribute 'TcIecLibraryType'}
	{attribute 'external_name' := 'F_VN_PadImageBorderExp_GUID_CD768495_4A48_45EA_D35A_6104A651B2F2'}
	(* Add padding around the original image borders. (expert function) *)
	FUNCTION F_VN_PadImageBorderExp : HRESULT
	VAR_INPUT
		ipSrcImage	:	ITcVnImage;	(* Source image *)
		ipPaddedImage	:	REFERENCE TO ITcVnImage;	(* Padded destination image (Same type as ipSrcImage, an appropriate destination image will be created if required.) *)
		nTopBorder	:	UDINT;	(* Padding height in pixels above top border *)
		nBottomBorder	:	UDINT;	(* Padding height in pixels below bottom border *)
		nLeftBorder	:	UDINT;	(* Padding width in pixels before left border *)
		nRightBorder	:	UDINT;	(* Padding width in pixels after right border *)
		ePaddingType	:	ETcVnBorderInterpolationMethod;	(* Specifies how the pixel values of the padding area are determined *)
	END_VAR
	VAR_IN_OUT
		aPaddingValue	:	TcVnVector4_LREAL;	(* Specifies the padding value if CONSTANT is used *)
	END_VAR
	VAR_INPUT
		hrPrev	:	HRESULT;	(* HRESULT indicating the result of previous operations (If SUCCEEDED(hrPrev) equals false, no operation is executed.) *)
	END_VAR

END_FUNCTION

// Functions/Machine Learning/F_VN_CreateBoostClassifier

	{attribute 'TcIecLibraryType'}
	{attribute 'external_name' := 'F_VN_CreateBoostClassifier_GUID_B6063C16_A11D_4814_D565_D627ED925C23'}
	(* Create a Boost classifier using the default parameters. The initial reference count is set to one if a new model is created and kept, otherwise. The Boost classifier is only applicable to binary classification problems. It learns to distinguish between samples labelled with two user-defined class labels by incrementally adding weak classifiers to improve the classification results. Models of this type neither support on-line training (sample by sample) nor retraining. *)
	FUNCTION F_VN_CreateBoostClassifier : HRESULT
	VAR_INPUT
		ipMlModel	:	REFERENCE TO ITcVnMlModel;	(* Returns the created model (Non-zero interface pointers are reused.) *)
		hrPrev	:	HRESULT;	(* HRESULT indicating the result of previous operations (If SUCCEEDED(hrPrev) equals false, no operation is executed.) *)
	END_VAR

END_FUNCTION

// Functions/Machine Learning/F_VN_CreateBoostClassifierExp

	{attribute 'TcIecLibraryType'}
	{attribute 'external_name' := 'F_VN_CreateBoostClassifierExp_GUID_B32382A8_407E_40B1_C0F7_1CBAAAECE683'}
	(* Create a Boost classifier. The initial reference count is set to one if a new model is created and kept, otherwise. The Boost classifier is only applicable to binary classification problems. It learns to distinguish between samples labelled with two user-defined class labels by incrementally adding weak classifiers to improve the classification results. Models of this type neither support on-line training (sample by sample) nor retraining. (expert function) *)
	FUNCTION F_VN_CreateBoostClassifierExp : HRESULT
	VAR_INPUT
		ipMlModel	:	REFERENCE TO ITcVnMlModel;	(* Returns the created model (Non-zero interface pointers are reused.) *)
		eType	:	ETcVnBoostClassifierType;	(* Learning algorithm type (default: TCVN_BCT_REAL) *)
		nMaxDepth	:	UDINT;	(* Maximum tree depth (default: 1) *)
		nMinSamples	:	UDINT;	(* Minimum number of samples within a node required for splitting (default: 10) *)
		nWeakClassifiers	:	UDINT;	(* Number of weak classifiers (default: 100) *)
		fWeightTrimRate	:	LREAL;	(* Weight threshold used during training (off: 0; default: 0.95). *)
		hrPrev	:	HRESULT;	(* HRESULT indicating the result of previous operations (If SUCCEEDED(hrPrev) equals false, no operation is executed.) *)
	END_VAR

END_FUNCTION

// Functions/Machine Learning/F_VN_CreateBoostClassifierExp2

	{attribute 'TcIecLibraryType'}
	{attribute 'external_name' := 'F_VN_CreateBoostClassifierExp2_GUID_073CFF09_AB37_4FAC_D2B3_5F913EB1A75C'}
	(* Create a Boost classifier. The initial reference count is set to one if a new model is created and kept, otherwise. The Boost classifier is only applicable to binary classification problems. It learns to distinguish between samples labelled with two user-defined class labels by incrementally adding weak classifiers to improve the classification results. Models of this type neither support on-line training (sample by sample) nor retraining. (expert function) *)
	FUNCTION F_VN_CreateBoostClassifierExp2 : HRESULT
	VAR_INPUT
		ipMlModel	:	REFERENCE TO ITcVnMlModel;	(* Returns the created model (Non-zero interface pointers are reused.) *)
		eType	:	ETcVnBoostClassifierType;	(* Learning algorithm type (default: TCVN_BCT_REAL) *)
		nMaxDepth	:	UDINT;	(* Maximum tree depth (default: 1) *)
		nMinSamples	:	UDINT;	(* Minimum number of samples within a node required for splitting (default: 10) *)
		nWeakClassifiers	:	UDINT;	(* Number of weak classifiers (default: 100) *)
		fWeightTrimRate	:	LREAL;	(* Weight threshold used during training (off: 0; default: 0.95). *)
		ipClassPriors	:	ITcVnContainer;	(* Class priors (ContainerType_Vector_REAL or ContainerType_Vector_LREAL; only for classifiers; optional, set to 0 if not required or not allowed; default: 0) *)
		hrPrev	:	HRESULT;	(* HRESULT indicating the result of previous operations (If SUCCEEDED(hrPrev) equals false, no operation is executed.) *)
	END_VAR

END_FUNCTION

// Functions/Machine Learning/F_VN_CreateKmppModel

	{attribute 'TcIecLibraryType'}
	{attribute 'external_name' := 'F_VN_CreateKmppModel_GUID_94A28DEF_889F_4799_EFE3_635BE42CA6C6'}
	(* Create a k-means++ model of the specified type. The initial reference count is set to one if a new model is created and kept, otherwise. Models of this type neither support on-line training (sample by sample) nor retraining. *)
	FUNCTION F_VN_CreateKmppModel : HRESULT
	VAR_INPUT
		ipMlModel	:	REFERENCE TO ITcVnMlModel;	(* Returns the created model (Non-zero interface pointers are reused.) *)
		eKmppType	:	ETcVnPrototypeClusterer;	(* k-means++ model type *)
		nK	:	UDINT;	(* Parameter k (number of clusters) *)
		hrPrev	:	HRESULT;	(* HRESULT indicating the result of previous operations (If SUCCEEDED(hrPrev) equals false, no operation is executed.) *)
	END_VAR

END_FUNCTION

// Functions/Machine Learning/F_VN_CreateKmppModelExp

	{attribute 'TcIecLibraryType'}
	{attribute 'external_name' := 'F_VN_CreateKmppModelExp_GUID_F9F44FC9_6C3D_48BA_C498_F76E7ACD64CE'}
	(* Create a k-means++ model of the specified type. The initial reference count is set to one if a new model is created and kept, otherwise. Models of this type neither support on-line training (sample by sample) nor retraining. (expert function) *)
	FUNCTION F_VN_CreateKmppModelExp : HRESULT
	VAR_INPUT
		ipMlModel	:	REFERENCE TO ITcVnMlModel;	(* Returns the created model (Non-zero interface pointers are reused.) *)
		eKmppType	:	ETcVnPrototypeClusterer;	(* k-means++ model type *)
		nK	:	UDINT;	(* Parameter k (number of clusters) *)
		bDoublePrecision	:	BOOL;	(* If true, the model is generated with double precision (LREAL) instead of single precision (REAL). (default: FALSE) *)
		nMaxIterations	:	UDINT;	(* Maximum number of iterations (triggers the usage of the default value of 10 if it equals 0) *)
		fEpsilon	:	LREAL;	(* Maximum allowed difference of the error between two successive iterations (triggers the usage of the default value of 0.001 if it equals 0) *)
		hrPrev	:	HRESULT;	(* HRESULT indicating the result of previous operations (If SUCCEEDED(hrPrev) equals false, no operation is executed.) *)
	END_VAR

END_FUNCTION

// Functions/Machine Learning/F_VN_CreateKnnModel

	{attribute 'TcIecLibraryType'}
	{attribute 'external_name' := 'F_VN_CreateKnnModel_GUID_5756F304_4FC0_4BA5_C53D_5AE362B8538E'}
	(* Create a k-nearest neighbors model of the specified type. The initial reference count is set to one if a new model is created and kept, otherwise. Models of this type support on-line training (sample by sample) and retraining. Predictions can only be scalar. *)
	FUNCTION F_VN_CreateKnnModel : HRESULT
	VAR_INPUT
		ipMlModel	:	REFERENCE TO ITcVnMlModel;	(* Returns the created model (Non-zero interface pointers are reused.) *)
		eKnnType	:	ETcVnKnn;	(* k-nearest neighbors model type *)
		nK	:	UDINT;	(* Parameter k used for prediction (number of considered neighbors) *)
		hrPrev	:	HRESULT;	(* HRESULT indicating the result of previous operations (If SUCCEEDED(hrPrev) equals false, no operation is executed.) *)
	END_VAR

END_FUNCTION

